	16#00000AD5:
		F_EtherCAT_VendorIDtoString := 'VA Laserautomation GmbH';

	16#00000AD6:
		F_EtherCAT_VendorIDtoString := 'Kleintges Elektrogeratebau GmbH';

	16#00000AD7:
		F_EtherCAT_VendorIDtoString := 'Logosol, Inc.';

	16#00000AD8:
		F_EtherCAT_VendorIDtoString := 'REJ Co., Ltd.';

	16#00000AD9:
		F_EtherCAT_VendorIDtoString := 'TCK Inc.';

	16#00000ADA:
		F_EtherCAT_VendorIDtoString := 'Axetris AG';

	16#00000ADB:
		F_EtherCAT_VendorIDtoString := 'Replicant Automation FZE';

	16#00000ADC:
		F_EtherCAT_VendorIDtoString := 'AIRTEC Pneumatic GmbH';

	16#00000ADD:
		F_EtherCAT_VendorIDtoString := 'Equip-Test Kft.';

	16#00000ADE:
		F_EtherCAT_VendorIDtoString := 'ChromaTan Corporation';

	16#00000ADF:
		F_EtherCAT_VendorIDtoString := 'Ford Motor Company Limited';

	16#00000AE0:
		F_EtherCAT_VendorIDtoString := 'thyssenkrupp Marine Systems GmbH';

	16#00000AE1:
		F_EtherCAT_VendorIDtoString := 'GEFAZ mbH';

	16#00000AE3:
		F_EtherCAT_VendorIDtoString := 'L&T Technology Services Limited';

	16#00000AE5:
		F_EtherCAT_VendorIDtoString := 'The Cyber University of Korea, Department of Mechanical and Control Engineering';

	16#00000AE6:
		F_EtherCAT_VendorIDtoString := 'SCHOBER Elektronik GmbH';

	16#00000AE7:
		F_EtherCAT_VendorIDtoString := 'Simulation and Control Technologies, Inc';

	16#00000AE8:
		F_EtherCAT_VendorIDtoString := 'Guangdong Sumida Automation Co.,Ltd.';

	16#00000AE9:
		F_EtherCAT_VendorIDtoString := 'GEMSS Medical Systems Co.,Ltd.';

	16#00000AEA:
		F_EtherCAT_VendorIDtoString := 'Shanghai Electric Power T&D Group';

	16#00000AEB:
		F_EtherCAT_VendorIDtoString := 'Shandong University, School of Control Science and Engineering';

	16#00000AEC:
		F_EtherCAT_VendorIDtoString := 'Fiessler Elektronik GmbH & Co. KG';

	16#00000AED:
		F_EtherCAT_VendorIDtoString := 'Cencorp Automation Technology Co, Ltd.';

	16#00000AEE:
		F_EtherCAT_VendorIDtoString := 'Venture International Pte Ltd';

	16#00000AEF:
		F_EtherCAT_VendorIDtoString := 'EcoTronic GmbH';

	16#00000AF0:
		F_EtherCAT_VendorIDtoString := 'Shenzhen Donglaier Smart Technology Co., Ltd.';

	16#00000AF1:
		F_EtherCAT_VendorIDtoString := 'Domino UK Limited';

	16#00000AF3:
		F_EtherCAT_VendorIDtoString := 'Elekta Solutions AB';

	16#00000AF4:
		F_EtherCAT_VendorIDtoString := 'Logic Fruit Technologies Pvt. Ltd.';

	16#00000AF5:
		F_EtherCAT_VendorIDtoString := 'ecocoach AG';

	16#00000AF6:
		F_EtherCAT_VendorIDtoString := 'SIOS Metechnik GmbH';

	16#00000AF7:
		F_EtherCAT_VendorIDtoString := 'Jabil Circuit Magyarorszag Kft.';

	16#00000AF8:
		F_EtherCAT_VendorIDtoString := 'seven dreamers laundroid, inc.';

	16#00000AF9:
		F_EtherCAT_VendorIDtoString := 'VR Group, a.s.';

	16#00000AFA:
		F_EtherCAT_VendorIDtoString := 'Afag Automation AG';

	16#00000AFB:
		F_EtherCAT_VendorIDtoString := 'Miyagi Nikon Precision Co., Ltd.';

	16#00000AFC:
		F_EtherCAT_VendorIDtoString := 'AutomationWare S.r.l.';

	16#00000AFD:
		F_EtherCAT_VendorIDtoString := 'Isar Aerospace Technologies GmbH';

	16#00000AFE:
		F_EtherCAT_VendorIDtoString := 'GTSystem GmbH';

	16#00000AFF:
		F_EtherCAT_VendorIDtoString := 'Technische Universitat Munchen, Department of Physics';

	16#00000B00:
		F_EtherCAT_VendorIDtoString := 'S+S Regeltechnik GmbH';

	16#00000B01:
		F_EtherCAT_VendorIDtoString := 'Osaka University, Graduate School of Engineering Science';

	16#00000B02:
		F_EtherCAT_VendorIDtoString := 'Vogtlin Instruments GmbH';

	16#00000B03:
		F_EtherCAT_VendorIDtoString := 'TOHAN DENSHI KIKI CO.,LTD.';

	16#00000B04:
		F_EtherCAT_VendorIDtoString := 'Shinwa Industries, Inc.';

	16#00000B05:
		F_EtherCAT_VendorIDtoString := 'Suzhou Linkhou Robot Co.,Ltd';

	16#00000B06:
		F_EtherCAT_VendorIDtoString := 'DMC, Inc.';

	16#00000B07:
		F_EtherCAT_VendorIDtoString := 'Nippon Pulse Motor Co., Ltd.';

	16#00000B08:
		F_EtherCAT_VendorIDtoString := 'LANG GmbH & Co. KG';

	16#00000B09:
		F_EtherCAT_VendorIDtoString := 'STICHT Technologie GmbH';

	16#00000B0A:
		F_EtherCAT_VendorIDtoString := 'HIMS Co., Ltd.';

	16#00000B0B:
		F_EtherCAT_VendorIDtoString := 'WITRON Logistik + Informatik GmbH';

	16#00000B0C:
		F_EtherCAT_VendorIDtoString := 'Vistec Electron Beam GmbH';

	16#00000B0D:
		F_EtherCAT_VendorIDtoString := 'General Atomics';

	16#00000B0E:
		F_EtherCAT_VendorIDtoString := 'Teubner Industrie-Elektronik GmbH';

	16#00000B0F:
		F_EtherCAT_VendorIDtoString := 'DEWETRON GmbH';

	16#00000B10:
		F_EtherCAT_VendorIDtoString := 'Philip Morris Products SA';

	16#00000B11:
		F_EtherCAT_VendorIDtoString := 'Nihon Protech Software Co., Ltd.';

	16#00000B13:
		F_EtherCAT_VendorIDtoString := 'Industrial Indexing Systems, Inc.';

	16#00000B14:
		F_EtherCAT_VendorIDtoString := 'AKIM METAL Sanayi Ve Ticaret Anonim Sirketi';

	16#00000B15:
		F_EtherCAT_VendorIDtoString := 'MEODAT Messtechnik, Ortung und Datenverarbeitung GmbH';

	16#00000B17:
		F_EtherCAT_VendorIDtoString := 'Goyo Electronics Co.,Ltd.';

	16#00000B18:
		F_EtherCAT_VendorIDtoString := 'Shanghai Golytec Automation Co., Ltd.';

	16#00000B19:
		F_EtherCAT_VendorIDtoString := 'Redcur GmbH';

	16#00000B1A:
		F_EtherCAT_VendorIDtoString := 'Room3327, Inc.';

	16#00000B1C:
		F_EtherCAT_VendorIDtoString := 'Love Electronics Ltd';

	16#00000B1D:
		F_EtherCAT_VendorIDtoString := 'Fontys University of Applied Sciences, School of Information & Communication Technology';

	16#00000B1E:
		F_EtherCAT_VendorIDtoString := 'Hocoma AG';

	16#00000B1F:
		F_EtherCAT_VendorIDtoString := 'Sensor Instruments Entwicklungs- und Vertriebs-GmbH';

	16#00000B20:
		F_EtherCAT_VendorIDtoString := 'Reboocon Bionics B.V.';

	16#00000B21:
		F_EtherCAT_VendorIDtoString := 'Evident Canada Inc.';

	16#00000B22:
		F_EtherCAT_VendorIDtoString := 'Photon Control Inc.';

	16#00000B23:
		F_EtherCAT_VendorIDtoString := 'NK Labs, LLC';

	16#00000B24:
		F_EtherCAT_VendorIDtoString := 'Excelpoint Systems (India) Pvt Ltd';

	16#00000B25:
		F_EtherCAT_VendorIDtoString := '"Gheorghe Asachi" Technical University of Iasi, Faculty of Automatic Control and Computer Engineering';

	16#00000B26:
		F_EtherCAT_VendorIDtoString := 'Manroland Sheetfed GmbH';

	16#00000B27:
		F_EtherCAT_VendorIDtoString := 'OPTEX FA CO., LTD.';

	16#00000B28:
		F_EtherCAT_VendorIDtoString := 'SMAC Corporation';

	16#00000B2A:
		F_EtherCAT_VendorIDtoString := 'SAITEL S.r.l.';

	16#00000B2B:
		F_EtherCAT_VendorIDtoString := 'Hebi Haichang Special Equipment Co.,Ltd.';

	16#00000B2C:
		F_EtherCAT_VendorIDtoString := 'Salunda Ltd';

	16#00000B2D:
		F_EtherCAT_VendorIDtoString := 'Higerman CNC Technology (SZ) Limited';

	16#00000B2E:
		F_EtherCAT_VendorIDtoString := 'IPG Laser GmbH & Co. KG';

	16#00000B2F:
		F_EtherCAT_VendorIDtoString := 'RTSoft, AO';

	16#00000B30:
		F_EtherCAT_VendorIDtoString := 'Dalian Hi-Sensor Technology Co., Ltd.';

	16#00000B31:
		F_EtherCAT_VendorIDtoString := 'alpiscan srls';

	16#00000B32:
		F_EtherCAT_VendorIDtoString := 'DYNAMIC OPTICS s.r.l.';

	16#00000B33:
		F_EtherCAT_VendorIDtoString := 'OOO “ITS-Sibir”';

	16#00000B34:
		F_EtherCAT_VendorIDtoString := 'SUMITOMO RIKO Company Limited';

	16#00000B35:
		F_EtherCAT_VendorIDtoString := 'Tianjin Automa Technology Co. Ltd.';

	16#00000B37:
		F_EtherCAT_VendorIDtoString := 'Human Automation Co., Ltd.';

	16#00000B38:
		F_EtherCAT_VendorIDtoString := 'Aplex Technology Inc.';

	16#00000B39:
		F_EtherCAT_VendorIDtoString := 'Shanghai Jesee Auto System Co., Ltd';

	16#00000B3A:
		F_EtherCAT_VendorIDtoString := 'Kunming Unionscience Technology Co.,Ltd';

	16#00000B3B:
		F_EtherCAT_VendorIDtoString := 'Fitz-Thors Engineering, Inc.';

	16#00000B3C:
		F_EtherCAT_VendorIDtoString := 'ACTIA Automotive SA';

	16#00000B3D:
		F_EtherCAT_VendorIDtoString := 'Kunshan SVL Electric Co.,Ltd';

	16#00000B3E:
		F_EtherCAT_VendorIDtoString := 'SilCore Technology';

	16#00000B3F:
		F_EtherCAT_VendorIDtoString := 'SHENZHEN QITAI TECHNOLOGY CO.LTD';

	16#00000B40:
		F_EtherCAT_VendorIDtoString := 'A. Sturzenegger Elektronik GmbH';

	16#00000B41:
		F_EtherCAT_VendorIDtoString := 'ZEUS CO., LTD.';

	16#00000B42:
		F_EtherCAT_VendorIDtoString := 'BETAMONT s.r.o.';

	16#00000B43:
		F_EtherCAT_VendorIDtoString := 'Strategy Automation S.r.l.';

	16#00000B44:
		F_EtherCAT_VendorIDtoString := 'Fachhochschule Nordwestschweiz, Hochschule fur Technik, Institut fur Automation';

	16#00000B45:
		F_EtherCAT_VendorIDtoString := 'SMS group GmbH';

	16#00000B46:
		F_EtherCAT_VendorIDtoString := 'TRUMPF Schweiz AG';

	16#00000B47:
		F_EtherCAT_VendorIDtoString := 'Fraunhofer-Institut fur Silicatforschung ISC';

	16#00000B48:
		F_EtherCAT_VendorIDtoString := 'The University of Tokyo, Graduate School of Information Science and Technology';

	16#00000B49:
		F_EtherCAT_VendorIDtoString := 'Indian Institute of Science, Interdisciplinary Centre for Energy Research';

	16#00000B4A:
		F_EtherCAT_VendorIDtoString := 'Overlay Technology OU';

	16#00000B4B:
		F_EtherCAT_VendorIDtoString := 'CK Automation, LLC';

	16#00000B4D:
		F_EtherCAT_VendorIDtoString := 'OOO "Kompex-T"';

	16#00000B4E:
		F_EtherCAT_VendorIDtoString := 'Ostbayerische Technische Hochschule Regensburg, Fakultat Maschinenbau';

	16#00000B4F:
		F_EtherCAT_VendorIDtoString := 'Hefei Eagle Automation Engineering Technology Co., Ltd.';

	16#00000B50:
		F_EtherCAT_VendorIDtoString := 'Vertiv Tech Co., Ltd';

	16#00000B51:
		F_EtherCAT_VendorIDtoString := 'Sanying MotionControl Instruments Ltd.';

	16#00000B52:
		F_EtherCAT_VendorIDtoString := 'Jiangsu Saiyang Mechanical & Electrical Technology Co., Ltd.';

	16#00000B53:
		F_EtherCAT_VendorIDtoString := 'Robosoft NV';

	16#00000B54:
		F_EtherCAT_VendorIDtoString := 'MotionBank';

	16#00000B55:
		F_EtherCAT_VendorIDtoString := 'South China University of Technology, School of Automation Science & Engineering';

	16#00000B56:
		F_EtherCAT_VendorIDtoString := 'Oetiker Schweiz AG';

	16#00000B57:
		F_EtherCAT_VendorIDtoString := 'Chiang Mai University, Faculty of Engineering';

	16#00000B58:
		F_EtherCAT_VendorIDtoString := 'Shenzhen FOXON Automation Technology Co., Ltd.';

	16#00000B59:
		F_EtherCAT_VendorIDtoString := 'Heinmade BV';

	16#00000B5A:
		F_EtherCAT_VendorIDtoString := 'ING-AUTOMATION';

	16#00000B5B:
		F_EtherCAT_VendorIDtoString := 'Vanteon Corporation';

	16#00000B5C:
		F_EtherCAT_VendorIDtoString := 'Solvine, Inc.';

	16#00000B5D:
		F_EtherCAT_VendorIDtoString := 'SHINWA Controls Co., Ltd.';

	16#00000B5E:
		F_EtherCAT_VendorIDtoString := 'Sierra CP Engineering Ltd.';

	16#00000B5F:
		F_EtherCAT_VendorIDtoString := 'Rope Robotics ApS';

	16#00000B60:
		F_EtherCAT_VendorIDtoString := 'Hefei Sineva Intelligent Machine Co.,Ltd';

	16#00000B61:
		F_EtherCAT_VendorIDtoString := 'Shenzhen Porcheson Technology Co., Ltd';

	16#00000B62:
		F_EtherCAT_VendorIDtoString := 'Greenlight Innovation Inc.';

	16#00000B63:
		F_EtherCAT_VendorIDtoString := 'PCB Piezotronics, Inc.';

	16#00000B64:
		F_EtherCAT_VendorIDtoString := 'microGauge AG';

	16#00000B65:
		F_EtherCAT_VendorIDtoString := 'EL Klaszter Iroda Kft.';

	16#00000B66:
		F_EtherCAT_VendorIDtoString := 'A.B.Esse Spa';

	16#00000B67:
		F_EtherCAT_VendorIDtoString := 'Corindus, Inc.';

	16#00000B68:
		F_EtherCAT_VendorIDtoString := 'Celeroton AG';

	16#00000B69:
		F_EtherCAT_VendorIDtoString := 'SAMHYUN Co. Ltd.';

	16#00000B6A:
		F_EtherCAT_VendorIDtoString := 'Ecole Polytechnique Federale de Lausanne, School of Basic Sciences';

	16#00000B6B:
		F_EtherCAT_VendorIDtoString := 'AVIC-XINHANG YUBEI STEERING SYSTEM (XINXIANG) CO.,LTD';

	16#00000B6C:
		F_EtherCAT_VendorIDtoString := 'Creative Conners, Inc.';

	16#00000B6D:
		F_EtherCAT_VendorIDtoString := 'Mamezou Co.,Ltd.';

	16#00000B6E:
		F_EtherCAT_VendorIDtoString := 'Raith B.V.';

	16#00000B6F:
		F_EtherCAT_VendorIDtoString := 'Soft Harmony';

	16#00000B70:
		F_EtherCAT_VendorIDtoString := 'Elektrik Uretim A.S.';

	16#00000B71:
		F_EtherCAT_VendorIDtoString := 'Delft University of Technology, Electronic and Mechanical Support Division (DEMO)';

	16#00000B72:
		F_EtherCAT_VendorIDtoString := 'machineering GmbH & Co. KG';

	16#00000B73:
		F_EtherCAT_VendorIDtoString := 'GRAPHIMECC S.r.l.';

	16#00000B74:
		F_EtherCAT_VendorIDtoString := 'TOPTICA Projects GmbH';

	16#00000B75:
		F_EtherCAT_VendorIDtoString := 'Enlaica Co., Ltd.';

	16#00000B76:
		F_EtherCAT_VendorIDtoString := 'SYSTEC Corporation';

	16#00000B77:
		F_EtherCAT_VendorIDtoString := 'Sherpa Inc.';

	16#00000B78:
		F_EtherCAT_VendorIDtoString := 'Sioux Embedded Systems B.V.';

	16#00000B79:
		F_EtherCAT_VendorIDtoString := 'UNISEM Co., Ltd.';

	16#00000B7A:
		F_EtherCAT_VendorIDtoString := 'William Petersen Elektronik A/S';

	16#00000B7B:
		F_EtherCAT_VendorIDtoString := 'Shanghai Velle Automobile Air Conditioner Co., Ltd.';

	16#00000B7C:
		F_EtherCAT_VendorIDtoString := 'Vision Tech Co.';

	16#00000B7D:
		F_EtherCAT_VendorIDtoString := 'Technische Universitat Wien, Fakultat fur Elektrotechnik und Informationstechnik';

	16#00000B7E:
		F_EtherCAT_VendorIDtoString := 'Universitat Augsburg, Fakultat fur Angewandte Informatik';

	16#00000B7F:
		F_EtherCAT_VendorIDtoString := 'Tecnomotion Srl';

	16#00000B80:
		F_EtherCAT_VendorIDtoString := 'Microservo Co., Ltd.';

	16#00000B81:
		F_EtherCAT_VendorIDtoString := 'Micro CleanRoom Technology GmbH';

	16#00000B82:
		F_EtherCAT_VendorIDtoString := 'Global Motion & Systems Inc.';

	16#00000B83:
		F_EtherCAT_VendorIDtoString := 'L3 Technologies, Datron Advanced Technologies';

	16#00000B84:
		F_EtherCAT_VendorIDtoString := 'NTN Technical Service Corporation';

	16#00000B85:
		F_EtherCAT_VendorIDtoString := 'Chugoku Electric Manufacturing Co.,Inc.';

	16#00000B86:
		F_EtherCAT_VendorIDtoString := 'European Spallation Source ERIC, Integrated Control System Division';

	16#00000B87:
		F_EtherCAT_VendorIDtoString := 'MARS CO., LTD.';

	16#00000B88:
		F_EtherCAT_VendorIDtoString := 'SCOPX LABS';

	16#00000B89:
		F_EtherCAT_VendorIDtoString := 'Laser Mechanisms, Inc.';

	16#00000B8A:
		F_EtherCAT_VendorIDtoString := 'TechnoPro, Inc.';

	16#00000B8B:
		F_EtherCAT_VendorIDtoString := 'Advanced Micro Controls, Inc.';

	16#00000B8C:
		F_EtherCAT_VendorIDtoString := 'Intelligence Technology of CEC Co., Ltd';

	16#00000B8D:
		F_EtherCAT_VendorIDtoString := 'Applied Dynamics International, Inc.';

	16#00000B8E:
		F_EtherCAT_VendorIDtoString := 'Conch Electronic Co.,Ltd.';

	16#00000B8F:
		F_EtherCAT_VendorIDtoString := 'Shenzhen Lisan M&E Co., Ltd.';

	16#00000B90:
		F_EtherCAT_VendorIDtoString := 'FOXIDE LLC';

	16#00000B91:
		F_EtherCAT_VendorIDtoString := 'C2P Inc.';

	16#00000B92:
		F_EtherCAT_VendorIDtoString := 'SonMicroSystem Co.';

	16#00000B94:
		F_EtherCAT_VendorIDtoString := 'HUST Automation System Co., Ltd.';

	16#00000B95:
		F_EtherCAT_VendorIDtoString := 'ASIX Electronics Corporation';

	16#00000B97:
		F_EtherCAT_VendorIDtoString := 'Laboratoire dAnalyse et dArchitecture des Systemes (LAAS-CNRS)';

	16#00000B98:
		F_EtherCAT_VendorIDtoString := 'KM DIGITECH CO., LTD.';

	16#00000B99:
		F_EtherCAT_VendorIDtoString := 'Sens4 A/S';

	16#00000B9A:
		F_EtherCAT_VendorIDtoString := 'Nidec Research and Development Center, Taiwan';

	16#00000B9D:
		F_EtherCAT_VendorIDtoString := 'Cajo Technologies Oy';

	16#00000B9E:
		F_EtherCAT_VendorIDtoString := 'VAS HIGH TECHNOLOGY SOLUTION CORPORATION';

	16#00000B9F:
		F_EtherCAT_VendorIDtoString := 'Beijing Chymotion Control Technology Co. Ltd';

	16#00000BA0:
		F_EtherCAT_VendorIDtoString := 'MarquipWardUnited';

	16#00000BA1:
		F_EtherCAT_VendorIDtoString := 'Komax Singapore Pte Ltd';

	16#00000BA2:
		F_EtherCAT_VendorIDtoString := 'Persimmon Technologies Corporation';

	16#00000BA3:
		F_EtherCAT_VendorIDtoString := 'Tohoku University, New Industry Creation Hatchery Center (NICHe), Fluctuation Free Facility (FFF)';

	16#00000BA4:
		F_EtherCAT_VendorIDtoString := 'Rheinische Fachhochschule Koln gGmbH, Ingenieurwesen';

	16#00000BA5:
		F_EtherCAT_VendorIDtoString := 'Luminize';

	16#00000BA6:
		F_EtherCAT_VendorIDtoString := 'v6e Limited';

	16#00000BA7:
		F_EtherCAT_VendorIDtoString := 'ECA ROBOTICS SASU';

	16#00000BA8:
		F_EtherCAT_VendorIDtoString := 'Sphere Fluidics Limited';

	16#00000BA9:
		F_EtherCAT_VendorIDtoString := 'WELCON Systems Inc.';

	16#00000BAA:
		F_EtherCAT_VendorIDtoString := 'Exor International S.p.A';

	16#00000BAB:
		F_EtherCAT_VendorIDtoString := 'Dekimo Turnhout';

	16#00000BAC:
		F_EtherCAT_VendorIDtoString := 'Lavender CE Pty Ltd';

	16#00000BAD:
		F_EtherCAT_VendorIDtoString := 'Science in Motion Technology Corporation, Ltd.';

	16#00000BAE:
		F_EtherCAT_VendorIDtoString := 'IST Ingenieurburo fur Sensortechnik GmbH';

	16#00000BAF:
		F_EtherCAT_VendorIDtoString := 'maku engineering GmbH';

	16#00000BB0:
		F_EtherCAT_VendorIDtoString := 'Geoservices Equipements SAS';

	16#00000BB1:
		F_EtherCAT_VendorIDtoString := 'NEST Electronics GmbH';

	16#00000BB2:
		F_EtherCAT_VendorIDtoString := 'MR Shim GmbH';

	16#00000BB4:
		F_EtherCAT_VendorIDtoString := 'Zettaone Technologies India Pvt Ltd';

	16#00000BB6:
		F_EtherCAT_VendorIDtoString := 'Universitat Augsburg, Fakultat fur angewandte Informatik, Institut fur Informatik';

	16#00000BB7:
		F_EtherCAT_VendorIDtoString := 'SCHUNK Electronic Solutions GmbH';

	16#00000BB8:
		F_EtherCAT_VendorIDtoString := 'KOORD Sarl';

	16#00000BB9:
		F_EtherCAT_VendorIDtoString := 'regenHU Ltd.';

	16#00000BBA:
		F_EtherCAT_VendorIDtoString := 'VONSCH spol. s r.o.';

	16#00000BBC:
		F_EtherCAT_VendorIDtoString := 'Bore Automation Tech. Co., Ltd.';

	16#00000BBD:
		F_EtherCAT_VendorIDtoString := 'Board Planning Co., Ltd.';

	16#00000BBE:
		F_EtherCAT_VendorIDtoString := 'Kamp & Kotter GmbH';

	16#00000BBF:
		F_EtherCAT_VendorIDtoString := 'IOTech Systems Limited';

	16#00000BC0:
		F_EtherCAT_VendorIDtoString := 'Altinay Robot Technologies Inc.';

	16#00000BC1:
		F_EtherCAT_VendorIDtoString := 'Lorenz Messtechnik GmbH';

	16#00000BC2:
		F_EtherCAT_VendorIDtoString := 'LJ Welding Automation';

	16#00000BC3:
		F_EtherCAT_VendorIDtoString := 'DMP Electronics Inc.';

	16#00000BC4:
		F_EtherCAT_VendorIDtoString := 'Dima Motor Tec. Co., Ltd.';

	16#00000BC5:
		F_EtherCAT_VendorIDtoString := 'Fraunhofer-Institut fur Produktionstechnik und Automatisierung';

	16#00000BC6:
		F_EtherCAT_VendorIDtoString := 'Schneider Electric (China) Co., Ltd.';

	16#00000BC7:
		F_EtherCAT_VendorIDtoString := 'Suzhou DaFang Special Vehicle Co., Ltd';

	16#00000BC8:
		F_EtherCAT_VendorIDtoString := 'Shenzhen OUYE Intelligent Technology Co., Ltd';

	16#00000BC9:
		F_EtherCAT_VendorIDtoString := 'HBH Microwave GmbH';

	16#00000BCA:
		F_EtherCAT_VendorIDtoString := 'MTA B.V.';

	16#00000BCB:
		F_EtherCAT_VendorIDtoString := 'SYSTEM ARTWARE, Inc.';

	16#00000BCC:
		F_EtherCAT_VendorIDtoString := 'ProDSP Technologies Zrt.';

	16#00000BCD:
		F_EtherCAT_VendorIDtoString := 'Hypersen Technologies Co., Ltd';

	16#00000BCE:
		F_EtherCAT_VendorIDtoString := 'Pyramid Vacuum LLC';

	16#00000BCF:
		F_EtherCAT_VendorIDtoString := 'Hanbaek Tech Co., Ltd.';

	16#00000BD0:
		F_EtherCAT_VendorIDtoString := 'SC3 Automation Inc.';

	16#00000BD1:
		F_EtherCAT_VendorIDtoString := 'Fachhochschule Nordwestschweiz, Hochschule fur Technik, Institut fur Sensorik und Elektronik';

	16#00000BD2:
		F_EtherCAT_VendorIDtoString := 'innofas GmbH';

	16#00000BD3:
		F_EtherCAT_VendorIDtoString := 'Orbray Co., Ltd.';

	16#00000BD4:
		F_EtherCAT_VendorIDtoString := 'YUNNAN KSEC INTELLIGENT EQUIPMENT CO.,LTD.';

	16#00000BD6:
		F_EtherCAT_VendorIDtoString := 'Industrial Solutions Zuid-Oost B.V. (Actemium Electronics)';

	16#00000BD7:
		F_EtherCAT_VendorIDtoString := 'BETONMAC S.A.';

	16#00000BD8:
		F_EtherCAT_VendorIDtoString := 'Manufacturing Objects';

	16#00000BD9:
		F_EtherCAT_VendorIDtoString := 'Chen Yuan International Co., Ltd.';

	16#00000BDB:
		F_EtherCAT_VendorIDtoString := 'Griffin Technology Co., Ltd.';

	16#00000BDC:
		F_EtherCAT_VendorIDtoString := 'RORZE CORPORATION';

	16#00000BDD:
		F_EtherCAT_VendorIDtoString := 'Bruker Daltonik GmbH';

	16#00000BDE:
		F_EtherCAT_VendorIDtoString := 'Logos01 Srl';

	16#00000BDF:
		F_EtherCAT_VendorIDtoString := 'Coaters Paradise GmbH';

	16#00000BE0:
		F_EtherCAT_VendorIDtoString := 'Hahn-Schickard-Gesellschaft fur angewandte Forschung e.V.';

	16#00000BE2:
		F_EtherCAT_VendorIDtoString := 'R&D Company "Vector" LLC';

	16#00000BE3:
		F_EtherCAT_VendorIDtoString := 'ReeR SpA';

	16#00000BE4:
		F_EtherCAT_VendorIDtoString := 'HP Scitex Ltd.';

	16#00000BE5:
		F_EtherCAT_VendorIDtoString := 'Hitachi Automotive Systems Americas, Inc.';

	16#00000BE6:
		F_EtherCAT_VendorIDtoString := 'Zhejiang Eternal Automation Sci-Tec Co.,Ltd';

	16#00000BE7:
		F_EtherCAT_VendorIDtoString := 'Shenzhen Siron Electrical Co.,Ltd.';

	16#00000BE8:
		F_EtherCAT_VendorIDtoString := 'ARUP Laboratories';

	16#00000BE9:
		F_EtherCAT_VendorIDtoString := 'LETech Co.,Ltd.';

	16#00000BEA:
		F_EtherCAT_VendorIDtoString := 'Bangkok University, School of Engineering, Robotics Laboratory';

	16#00000BEB:
		F_EtherCAT_VendorIDtoString := 'Kontron Electronics GmbH';

	16#00000BEC:
		F_EtherCAT_VendorIDtoString := 'Shanghai Junqian Sensing Technology Co., Ltd.';

	16#00000BEE:
		F_EtherCAT_VendorIDtoString := 'VI.BE.MAC s.p.a.';

	16#00000BEF:
		F_EtherCAT_VendorIDtoString := 'EMG Automation GmbH';

	16#00000BF0:
		F_EtherCAT_VendorIDtoString := 'American Controls & Automation, Inc.';

	16#00000BF1:
		F_EtherCAT_VendorIDtoString := 'Ascale Enterprise Co., Ltd.';

	16#00000BF2:
		F_EtherCAT_VendorIDtoString := 'University of Applied Sciences and Arts Western Switzerland (HES-SO Fribourg)';

	16#00000BF3:
		F_EtherCAT_VendorIDtoString := 'Lantronix, Inc.';

	16#00000BF4:
		F_EtherCAT_VendorIDtoString := 'Technische Hochschule Rosenheim';

	16#00000BF5:
		F_EtherCAT_VendorIDtoString := 'LEIFERT INDUCTION GmbH';

	16#00000BF6:
		F_EtherCAT_VendorIDtoString := 'Automation of Things Europe GmbH';

	16#00000BF7:
		F_EtherCAT_VendorIDtoString := 'SAMWON ACT Co.,Ltd';

	16#00000BF8:
		F_EtherCAT_VendorIDtoString := 'Wenling Yuhai Electromechanical CO.,LTD';

	16#00000BF9:
		F_EtherCAT_VendorIDtoString := 'Faraday Motion Controls Ltd.';

	16#00000BFA:
		F_EtherCAT_VendorIDtoString := 'Nikon Systems Inc.';

	16#00000BFB:
		F_EtherCAT_VendorIDtoString := 'Sanitas EG S.r.l.';

	16#00000BFC:
		F_EtherCAT_VendorIDtoString := 'Videojet Technologies Inc.';

	16#00000BFD:
		F_EtherCAT_VendorIDtoString := 'ABB AG';

	16#00000BFE:
		F_EtherCAT_VendorIDtoString := 'WARDJet LLC';

	16#00000BFF:
		F_EtherCAT_VendorIDtoString := 'Ichor Systems, Inc.';

	16#00000C00:
		F_EtherCAT_VendorIDtoString := 'UTAREX Co., Ltd.';

	16#00000C01:
		F_EtherCAT_VendorIDtoString := 'GAON SOLUTION Ltd.';

	16#00000C02:
		F_EtherCAT_VendorIDtoString := 'Highlight Tech Corp.';

	16#00000C03:
		F_EtherCAT_VendorIDtoString := 'PO OWEN LLC';

	16#00000C04:
		F_EtherCAT_VendorIDtoString := 'RFPT Co., Ltd.';

	16#00000C05:
		F_EtherCAT_VendorIDtoString := 'Roboteq, Inc.';

	16#00000C06:
		F_EtherCAT_VendorIDtoString := 'Norgren Manufacturing Co., Ltd.';

	16#00000C07:
		F_EtherCAT_VendorIDtoString := 'FarmWise Labs, Inc.';

	16#00000C08:
		F_EtherCAT_VendorIDtoString := 'AŽD Praha s.r.o.';

	16#00000C0A:
		F_EtherCAT_VendorIDtoString := 'Can Man AG';

	16#00000C0B:
		F_EtherCAT_VendorIDtoString := 'Plustherm Point AG';

	16#00000C0C:
		F_EtherCAT_VendorIDtoString := 'MinebeaMitsumi Inc.';

	16#00000C0D:
		F_EtherCAT_VendorIDtoString := 'System Level Solutions (India) Pvt. Ltd.';

	16#00000C0E:
		F_EtherCAT_VendorIDtoString := 'EverMAX s.r.o.';

	16#00000C0F:
		F_EtherCAT_VendorIDtoString := 'Maruyama Manufacturing Corporation (DBA Maruyama Chillers Corporation)';

	16#00000C10:
		F_EtherCAT_VendorIDtoString := 'Han’s Assembly and Testing Technology (Singapore) Pte. Ltd.';

	16#00000C11:
		F_EtherCAT_VendorIDtoString := 'Cordova Industrial Integradores S.A. de C.V.';

	16#00000C12:
		F_EtherCAT_VendorIDtoString := 'NAMOO Co., Ltd.';

	16#00000C13:
		F_EtherCAT_VendorIDtoString := 'Blu Technology di Ing Carlo Mauri';

	16#00000C14:
		F_EtherCAT_VendorIDtoString := 'isel Germany AG';

	16#00000C15:
		F_EtherCAT_VendorIDtoString := 'UNITEK Industrie Elektronik GmbH';

	16#00000C16:
		F_EtherCAT_VendorIDtoString := 'Tohan-Engineering Corporation';

	16#00000C17:
		F_EtherCAT_VendorIDtoString := 'Machine Prognostics AS';

	16#00000C18:
		F_EtherCAT_VendorIDtoString := 'Avestron Inc.';

	16#00000C19:
		F_EtherCAT_VendorIDtoString := 'AP Systems Co., Ltd.';

	16#00000C1A:
		F_EtherCAT_VendorIDtoString := 'TIAN JIN SUNKE DIGITAL CONTROL TECHNOLOGY CO.,LTD';

	16#00000C1B:
		F_EtherCAT_VendorIDtoString := 'Robotech Co., Ltd.';

	16#00000C1C:
		F_EtherCAT_VendorIDtoString := 'AccuteX Technologies Co., Ltd.';

	16#00000C1D:
		F_EtherCAT_VendorIDtoString := 'Coherent Mainz (DILAS Diodenlaser GmbH)';

	16#00000C1E:
		F_EtherCAT_VendorIDtoString := 'Daxta Equipamentos Eletronicos Industria e Comercio Ltda';

	16#00000C20:
		F_EtherCAT_VendorIDtoString := 'ADG Automatisierung Dresden GmbH';

	16#00000C21:
		F_EtherCAT_VendorIDtoString := 'WHITEvoid GmbH';

	16#00000C22:
		F_EtherCAT_VendorIDtoString := 'BAS BV';

	16#00000C23:
		F_EtherCAT_VendorIDtoString := 'RS Elektroniksysteme GmbH';

	16#00000C25:
		F_EtherCAT_VendorIDtoString := 'HORIBA FuelCon GmbH';

	16#00000C26:
		F_EtherCAT_VendorIDtoString := 'miCos Iberia S.L.';

	16#00000C27:
		F_EtherCAT_VendorIDtoString := 'Slovak Academy of Sciences, Institute of Electrical Engineering';

	16#00000C28:
		F_EtherCAT_VendorIDtoString := 'Roketsan A.S.';

	16#00000C29:
		F_EtherCAT_VendorIDtoString := 'Bescom Global Co., Ltd.';

	16#00000C2A:
		F_EtherCAT_VendorIDtoString := 'Magnet-Schultz GmbH & Co. KG';

	16#00000C2B:
		F_EtherCAT_VendorIDtoString := 'NEWSUBSTANCE Limited';

	16#00000C2C:
		F_EtherCAT_VendorIDtoString := 'JingQi (Tianjin) Technology Co., Ltd.';

	16#00000C2D:
		F_EtherCAT_VendorIDtoString := 'TSK Prufsysteme GmbH';

	16#00000C2E:
		F_EtherCAT_VendorIDtoString := 'Airity Technologies, Inc.';

	16#00000C2F:
		F_EtherCAT_VendorIDtoString := 'EEP Elektro Elektronik Pranjic GmbH';

	16#00000C30:
		F_EtherCAT_VendorIDtoString := 'MovekoTech Oy';

	16#00000C31:
		F_EtherCAT_VendorIDtoString := 'Federal State Institution "Scientific Research Institute for System Analysis of the Russian Academy of Sciences"';

	16#00000C32:
		F_EtherCAT_VendorIDtoString := 'Nearfield Instruments B.V.';

	16#00000C33:
		F_EtherCAT_VendorIDtoString := 'TUBITAK BILGEM, National Research Institute of Electronics and Cryptology (UEKAE)';

	16#00000C34:
		F_EtherCAT_VendorIDtoString := 'Siemens Energy Global GmbH & Co. KG';

	16#00000C35:
		F_EtherCAT_VendorIDtoString := 'progress Maschinen & Automation AG';

	16#00000C36:
		F_EtherCAT_VendorIDtoString := 'Heliotis AG';

	16#00000C37:
		F_EtherCAT_VendorIDtoString := 'Strong Plus Technology GmbH';

	16#00000C38:
		F_EtherCAT_VendorIDtoString := 'LS Energy Solutions LLC';

	16#00000C39:
		F_EtherCAT_VendorIDtoString := 'Yaskawa Controls Co., Ltd.';

	16#00000C3A:
		F_EtherCAT_VendorIDtoString := 'NOVUSS-Automation GmbH';

	16#00000C3C:
		F_EtherCAT_VendorIDtoString := 'Sanwa Engineering Corp.';

	16#00000C3D:
		F_EtherCAT_VendorIDtoString := 'WIBOND Informationssysteme GmbH';

	16#00000C3E:
		F_EtherCAT_VendorIDtoString := 'MSP, a division of TSI Inc.';

	16#00000C3F:
		F_EtherCAT_VendorIDtoString := 'Wuxi Xinchang Electronic Technology Co., Ltd.';

	16#00000C40:
		F_EtherCAT_VendorIDtoString := 'NDK Semiconductor Co., Ltd.';

	16#00000C41:
		F_EtherCAT_VendorIDtoString := 'MS Ultraschall Technologie GmbH';

	16#00000C42:
		F_EtherCAT_VendorIDtoString := 'Korea University of Technology and Education (KOREATECH)';

	16#00000C43:
		F_EtherCAT_VendorIDtoString := 'Accelerated Software Engineering Ltd.';

	16#00000C44:
		F_EtherCAT_VendorIDtoString := 'Shenzhen Instar Electromechanical Technology Development Co., Ltd.';

	16#00000C45:
		F_EtherCAT_VendorIDtoString := 'Redler Technologies Ltd.';

	16#00000C46:
		F_EtherCAT_VendorIDtoString := 'NPOOO "Sital"';

	16#00000C47:
		F_EtherCAT_VendorIDtoString := 'Eaton Corporation';

	16#00000C48:
		F_EtherCAT_VendorIDtoString := 'Techservo (Shenzhen) Co., Ltd.';

	16#00000C49:
		F_EtherCAT_VendorIDtoString := 'Fabmatics GmbH';

	16#00000C4A:
		F_EtherCAT_VendorIDtoString := 'Sasaki Sekkei Co., Ltd.';

	16#00000C4B:
		F_EtherCAT_VendorIDtoString := 'Lohnert Elektronik GmbH';

	16#00000C4C:
		F_EtherCAT_VendorIDtoString := 'Vendee Concept SA';

	16#00000C4D:
		F_EtherCAT_VendorIDtoString := 'Nobleo Technology Holding BV';

	16#00000C4E:
		F_EtherCAT_VendorIDtoString := 'ECI Technology, Inc.';

	16#00000C4F:
		F_EtherCAT_VendorIDtoString := 'Linus G Productions GmbH';

	16#00000C50:
		F_EtherCAT_VendorIDtoString := 'PCB Elektronik San. Ve Tic. Ltd. Sti.';

	16#00000C51:
		F_EtherCAT_VendorIDtoString := 'Omron Scientific Technologies, Inc.';

	16#00000C52:
		F_EtherCAT_VendorIDtoString := 'Engineered Arts Limited';

	16#00000C53:
		F_EtherCAT_VendorIDtoString := 'NASA Jet Propulsion Laboratory';

	16#00000C54:
		F_EtherCAT_VendorIDtoString := 'Accelovant Technologies Corporation';

	16#00000C55:
		F_EtherCAT_VendorIDtoString := 'Hirata Corporation';

	16#00000C56:
		F_EtherCAT_VendorIDtoString := 'Fujian Nebula Electronics Co.,Ltd.';

	16#00000C57:
		F_EtherCAT_VendorIDtoString := 'Test Research, Inc.';

	16#00000C58:
		F_EtherCAT_VendorIDtoString := 'CYSCO Co., Ltd.';

	16#00000C59:
		F_EtherCAT_VendorIDtoString := 'Esko-Graphics Kongsberg AS';

	16#00000C5A:
		F_EtherCAT_VendorIDtoString := 'WOT Co.,Ltd.';

	16#00000C5C:
		F_EtherCAT_VendorIDtoString := 'SHENZHEN SENMUN ELECTRICAL CO.,LTD';

	16#00000C5D:
		F_EtherCAT_VendorIDtoString := 'Izhprest Ltd.';

	16#00000C5E:
		F_EtherCAT_VendorIDtoString := 'HAWE Hydraulik SE';

	16#00000C5F:
		F_EtherCAT_VendorIDtoString := 'Finetech GmbH & Co. KG';

	16#00000C60:
		F_EtherCAT_VendorIDtoString := 'Mitutoyo Corporation';

	16#00000C61:
		F_EtherCAT_VendorIDtoString := 'Cremer Speciaalmachines B.V.';

	16#00000C62:
		F_EtherCAT_VendorIDtoString := 'Astec Co., Ltd.';

	16#00000C64:
		F_EtherCAT_VendorIDtoString := 'ELNA LTD.';

	16#00000C65:
		F_EtherCAT_VendorIDtoString := 'Janasi Industries Ltd.';

	16#00000C66:
		F_EtherCAT_VendorIDtoString := 'Universidad de La Frontera, Facultad de Ingenieria y Ciencias, Centro de Modelacion y Computacion Cientifica (CEMCC)';

	16#00000C67:
		F_EtherCAT_VendorIDtoString := 'KALEJA GmbH';

	16#00000C68:
		F_EtherCAT_VendorIDtoString := 'Caldwell Machines & Tools trading as CMT Engineering';

	16#00000C69:
		F_EtherCAT_VendorIDtoString := 'ILJIN Global Holdings Co., Ltd.';

	16#00000C6A:
		F_EtherCAT_VendorIDtoString := 'Proteus Vietnam Limited';

	16#00000C6C:
		F_EtherCAT_VendorIDtoString := 'JUKI CORPORATION';

	16#00000C6D:
		F_EtherCAT_VendorIDtoString := 'MT Drive & Control (Shenzhen) Co.,Ltd';

	16#00000C6E:
		F_EtherCAT_VendorIDtoString := 'ShenZhen HongChuangXing Motion Technology Co.,Ltd';

	16#00000C6F:
		F_EtherCAT_VendorIDtoString := 'isMedia Co., Ltd.';

	16#00000C70:
		F_EtherCAT_VendorIDtoString := 'Shenzhen Yangshun Tongda Digital Technology Co., Ltd.';

	16#00000C71:
		F_EtherCAT_VendorIDtoString := 'MVTECH Co.,Ltd.';

	16#00000C72:
		F_EtherCAT_VendorIDtoString := 'Kane Terry Partridge dba Open Designer';

	16#00000C73:
		F_EtherCAT_VendorIDtoString := 'EK-Electronics GmbH';

	16#00000C74:
		F_EtherCAT_VendorIDtoString := 'Jiann Sheng Machinery & Electric Industrial Co., Ltd';

	16#00000C75:
		F_EtherCAT_VendorIDtoString := 'Gable Systems B.V.';

	16#00000C76:
		F_EtherCAT_VendorIDtoString := 'Constructions-3D SAS';

	16#00000C77:
		F_EtherCAT_VendorIDtoString := 'MIP robotics';

	16#00000C78:
		F_EtherCAT_VendorIDtoString := 'YouTool Automation Co., Ltd.';

	16#00000C79:
		F_EtherCAT_VendorIDtoString := 'Nanjing WEILAN Intelligent Technologies Co., Ltd.';

	16#00000C7A:
		F_EtherCAT_VendorIDtoString := 'ABB S.p.A.';

	16#00000C7B:
		F_EtherCAT_VendorIDtoString := 'Typhoon HIL Inc.';

	16#00000C7C:
		F_EtherCAT_VendorIDtoString := 'BLUTek Inc.';

	16#00000C7D:
		F_EtherCAT_VendorIDtoString := 'University of Engineering and Technology, Lahore, Al-Khwarizmi Institute of Computer Science, Human-Centered Robotics Lab';

	16#00000C7E:
		F_EtherCAT_VendorIDtoString := 'Technische Universitat Munchen, Fakultat fur Informatik, Lehrstuhl fur Robotik, Kunstliche Intelligenz und Echtzeitsysteme (Informatik 6)';

	16#00000C7F:
		F_EtherCAT_VendorIDtoString := 'Northrop Grumman Sperry Marine B.V. German Branch';

	16#00000C80:
		F_EtherCAT_VendorIDtoString := 'Technical University of Munich, Department of Electrical and Computer Engineering, Institute for Cognitive Systems (ICS)';

	16#00000C81:
		F_EtherCAT_VendorIDtoString := 'TNO';

	16#00000C82:
		F_EtherCAT_VendorIDtoString := 'IK Electronic Manufacturing Services S.L.U';

	16#00000C83:
		F_EtherCAT_VendorIDtoString := 'Ningbo Schleicher Technology Group Co., Ltd.';

	16#00000C84:
		F_EtherCAT_VendorIDtoString := 'TOWA Corporation';

	16#00000C85:
		F_EtherCAT_VendorIDtoString := 'Amacker Automation';

	16#00000C86:
		F_EtherCAT_VendorIDtoString := 'Hardt B.V.';

	16#00000C87:
		F_EtherCAT_VendorIDtoString := 'Anurichip System Inc.';

	16#00000C88:
		F_EtherCAT_VendorIDtoString := 'MESCO Engineering GmbH';

	16#00000C89:
		F_EtherCAT_VendorIDtoString := 'Oki Electric Industry Co., Ltd.';

	16#00000C8A:
		F_EtherCAT_VendorIDtoString := 'Motorsports Electronics, LLC';

	16#00000C8B:
		F_EtherCAT_VendorIDtoString := 'PPT Co., Ltd.';

	16#00000C8C:
		F_EtherCAT_VendorIDtoString := 'KYEONGIN TECH Co., Ltd.';

	16#00000C8D:
		F_EtherCAT_VendorIDtoString := 'SAS GYS';

	16#00000C8E:
		F_EtherCAT_VendorIDtoString := 'Cyber Surgery S.L.';

	16#00000C8F:
		F_EtherCAT_VendorIDtoString := 'CASTEK Mechatron Ind Co., Ltd.';

	16#00000C90:
		F_EtherCAT_VendorIDtoString := 'ERMAKSAN MAKINA SANAYI VE TICARET A.S.';

	16#00000C91:
		F_EtherCAT_VendorIDtoString := 'Elbit Systems Land Ltd.';

	16#00000C93:
		F_EtherCAT_VendorIDtoString := 'Javox Solutions GmbH';

	16#00000C94:
		F_EtherCAT_VendorIDtoString := 'Resilient Power Systems, Inc.';

	16#00000C95:
		F_EtherCAT_VendorIDtoString := 'CMRO Engineering';

	16#00000C96:
		F_EtherCAT_VendorIDtoString := 'Teknic, Inc.';

	16#00000C97:
		F_EtherCAT_VendorIDtoString := 'Lug Healthcare Technology S.L.';

	16#00000C98:
		F_EtherCAT_VendorIDtoString := 'Michael Koch GmbH';

	16#00000C99:
		F_EtherCAT_VendorIDtoString := 'UEC Scientific Instrument Co., Ltd.';

	16#00000C9A:
		F_EtherCAT_VendorIDtoString := 'WEISS GmbH';

	16#00000C9B:
		F_EtherCAT_VendorIDtoString := 'NITTOSEIKO CO., LTD.';

	16#00000C9C:
		F_EtherCAT_VendorIDtoString := 'WANTS Inc.';

	16#00000C9D:
		F_EtherCAT_VendorIDtoString := 'Tecnosens S.p.A.';

	16#00000C9F:
		F_EtherCAT_VendorIDtoString := 'Print Web International, Inc.';

	16#00000CA0:
		F_EtherCAT_VendorIDtoString := 'FAIR Innovation(Suzhou) Robot System Co.,Ltd.';

	16#00000CA1:
		F_EtherCAT_VendorIDtoString := 'OptiViz Technology, Inc.';

	16#00000CA2:
		F_EtherCAT_VendorIDtoString := 'Shanghai YISU Information Technologies Co.,Ltd.';

	16#00000CA3:
		F_EtherCAT_VendorIDtoString := 'Re S.p.A. Controlli Industriali';

	16#00000CA4:
		F_EtherCAT_VendorIDtoString := 'Canon Medical Systems Corporation';

	16#00000CA5:
		F_EtherCAT_VendorIDtoString := 'Suzhou Geyuan Electric Co., Ltd.';

	16#00000CA6:
		F_EtherCAT_VendorIDtoString := 'Shenzhen MICFIND Drive Technology Co., Ltd.';

	16#00000CA7:
		F_EtherCAT_VendorIDtoString := 'SECOM SRL';

	16#00000CA8:
		F_EtherCAT_VendorIDtoString := 'Panasonic Connect Co., Ltd.';

	16#00000CA9:
		F_EtherCAT_VendorIDtoString := 'BeiJing Agile Robots Technology Co.,Ltd.';

	16#00000CAB:
		F_EtherCAT_VendorIDtoString := 'Taiwan Innovative Space, Inc.';

	16#00000CAC:
		F_EtherCAT_VendorIDtoString := 'ABB Technikerschule';

	16#00000CAD:
		F_EtherCAT_VendorIDtoString := 'NOMOS Srl Tecnologie del Software';

	16#00000CAF:
		F_EtherCAT_VendorIDtoString := 'JSCC AUTOMATION (XIAMEN) LTD.';

	16#00000CB0:
		F_EtherCAT_VendorIDtoString := 'GMVT GmbH';

	16#00000CB1:
		F_EtherCAT_VendorIDtoString := 'Swisslog AG';

	16#00000CB2:
		F_EtherCAT_VendorIDtoString := 'Therm-x of California Inc.';

	16#00000CB3:
		F_EtherCAT_VendorIDtoString := 'CogniMade s.r.l.';

	16#00000CB4:
		F_EtherCAT_VendorIDtoString := 'SERT METAL SAS';

	16#00000CB5:
		F_EtherCAT_VendorIDtoString := 'Kardanan Shargh Co.';

	16#00000CB6:
		F_EtherCAT_VendorIDtoString := 'MPEX ROBOTICS KFT.';

	16#00000CB7:
		F_EtherCAT_VendorIDtoString := 'Critical Link LLC';

	16#00000CB8:
		F_EtherCAT_VendorIDtoString := 'Flokontrol Endustriyel Otomasyon San. ve Tic. Koll. Sti.';

	16#00000CB9:
		F_EtherCAT_VendorIDtoString := 'Nidec Avtron Automation Corporation';

	16#00000CBA:
		F_EtherCAT_VendorIDtoString := 'Alphasystem Co.,Ltd.';

	16#00000CBB:
		F_EtherCAT_VendorIDtoString := 'Carendes BVBA';

	16#00000CBC:
		F_EtherCAT_VendorIDtoString := 'Eltorque AS';

	16#00000CBD:
		F_EtherCAT_VendorIDtoString := 'University of Alberta, Faculty of Engineering';

	16#00000CBE:
		F_EtherCAT_VendorIDtoString := 'TOSIL Systems Private Limited';

	16#00000CBF:
		F_EtherCAT_VendorIDtoString := 'DELTA I/O CO.,LTD';

	16#00000CC0:
		F_EtherCAT_VendorIDtoString := 'Sipronika d.o.o.';

	16#00000CC1:
		F_EtherCAT_VendorIDtoString := 'TESA SARL';

	16#00000CC2:
		F_EtherCAT_VendorIDtoString := 'NXP B.V.';

	16#00000CC3:
		F_EtherCAT_VendorIDtoString := 'HERMOS AG';

	16#00000CC4:
		F_EtherCAT_VendorIDtoString := 'Svaya Robotics Pvt. Ltd.';

	16#00000CC5:
		F_EtherCAT_VendorIDtoString := 'ARRIVAL LTD.';

	16#00000CC6:
		F_EtherCAT_VendorIDtoString := 'Mold-Masters (2007) Limited';

	16#00000CC8:
		F_EtherCAT_VendorIDtoString := 'Hypex, d.o.o.';

	16#00000CC9:
		F_EtherCAT_VendorIDtoString := 'Sansei Technologies, Inc.';

	16#00000CCA:
		F_EtherCAT_VendorIDtoString := 'Shanghai United Imaging Healthcare Co., Ltd.';

	16#00000CCB:
		F_EtherCAT_VendorIDtoString := 'Seoul National University';

	16#00000CCC:
		F_EtherCAT_VendorIDtoString := '3C MACHINERY CO.,LTD.';

	16#00000CCD:
		F_EtherCAT_VendorIDtoString := 'CHINO CORPORATION';

	16#00000CCE:
		F_EtherCAT_VendorIDtoString := 'WUHAN MOTUS TECH CO.,LTD.';

	16#00000CCF:
		F_EtherCAT_VendorIDtoString := 'TPC Mechatronics Corp.';

	16#00000CD0:
		F_EtherCAT_VendorIDtoString := 'Philips Medical Systems DMC GmbH';

	16#00000CD1:
		F_EtherCAT_VendorIDtoString := 'TAZMO Co., Ltd.';

	16#00000CD2:
		F_EtherCAT_VendorIDtoString := 'Robo-Technology GmbH';

	16#00000CD3:
		F_EtherCAT_VendorIDtoString := 'Vivo Surgical Private Limited';

	16#00000CD4:
		F_EtherCAT_VendorIDtoString := 'Defence Research and Development Organisation, Research & Development Establishment (Engineers)';

	16#00000CD5:
		F_EtherCAT_VendorIDtoString := 'Jiangsu Shenzhou Semiconductor Technology Co., Ltd.';

	16#00000CD6:
		F_EtherCAT_VendorIDtoString := 'GrainSoft';

	16#00000CD7:
		F_EtherCAT_VendorIDtoString := 'MECCAD Sarl';

	16#00000CD9:
		F_EtherCAT_VendorIDtoString := 'National Formosa University, Department of Aeronautical Engineering, Innovative Design and Energy Application Lab. (IDEALab)';

	16#00000CDA:
		F_EtherCAT_VendorIDtoString := 'TOS Inc.';

	16#00000CDB:
		F_EtherCAT_VendorIDtoString := 'GTM Testing and Metrology GmbH';

	16#00000CDC:
		F_EtherCAT_VendorIDtoString := 'Prvni Signalni, a.s.';

	16#00000CDD:
		F_EtherCAT_VendorIDtoString := 'Georgia Institute of Technology, ECE Department, Center for Distributed Energy (CDE)';

	16#00000CDE:
		F_EtherCAT_VendorIDtoString := 'Plexim GmbH';

	16#00000CDF:
		F_EtherCAT_VendorIDtoString := 'Automation Industrial, Inc.';

	16#00000CE0:
		F_EtherCAT_VendorIDtoString := 'Regloplas AG';

	16#00000CE1:
		F_EtherCAT_VendorIDtoString := 'Azureus Solutions Ltd';

	16#00000CE2:
		F_EtherCAT_VendorIDtoString := 'Safran Electronics & Defense SAS';

	16#00000CE3:
		F_EtherCAT_VendorIDtoString := 'Sogeti Nederland B.V.';

	16#00000CE4:
		F_EtherCAT_VendorIDtoString := 'AKRYVIA SAS';

	16#00000CE5:
		F_EtherCAT_VendorIDtoString := 'FIRSTEC CO.,LTD.';

	16#00000CE6:
		F_EtherCAT_VendorIDtoString := 'M.D. Micro Detectors S.p.A.';

	16#00000CE7:
		F_EtherCAT_VendorIDtoString := 'Dataletics GmbH';

	16#00000CE8:
		F_EtherCAT_VendorIDtoString := 'Korea Institute of Machinery & Materials, Advanced Manufacturing Systems Research Division, Department of Ultra-Precision Machines and Systems';

	16#00000CE9:
		F_EtherCAT_VendorIDtoString := 'AEG Identifikationssysteme GmbH';

	16#00000CEA:
		F_EtherCAT_VendorIDtoString := 'CEA LIST';

	16#00000CEB:
		F_EtherCAT_VendorIDtoString := 'Shenyang Siasun Digital Drive Co., Ltd.';

	16#00000CEC:
		F_EtherCAT_VendorIDtoString := 'TissUse GmbH';

	16#00000CED:
		F_EtherCAT_VendorIDtoString := 'LithExx-Systems GmbH';

	16#00000CEE:
		F_EtherCAT_VendorIDtoString := 'AICRA s.r.o.';

	16#00000CEF:
		F_EtherCAT_VendorIDtoString := 'JANOME Corporation';

	16#00000CF0:
		F_EtherCAT_VendorIDtoString := 'Cambridge Filter Corporation';

	16#00000CF2:
		F_EtherCAT_VendorIDtoString := 'Celox Photonics Technology Inc.';

	16#00000CF3:
		F_EtherCAT_VendorIDtoString := 'swissQprint AG';

	16#00000CF4:
		F_EtherCAT_VendorIDtoString := 'COMFILE Technology INC.';

	16#00000CF5:
		F_EtherCAT_VendorIDtoString := 'Chengdu Vantron Technology Co., Ltd.';

	16#00000CF6:
		F_EtherCAT_VendorIDtoString := 'Duale Hochschule Baden-Wurttemberg Mannheim, Fakultat Technik, Studiengang Elektrotechnik';

	16#00000CF7:
		F_EtherCAT_VendorIDtoString := 'Tesollo Inc.';

	16#00000CF8:
		F_EtherCAT_VendorIDtoString := 'Roundpeg Technologies GmbH';

	16#00000CF9:
		F_EtherCAT_VendorIDtoString := 'Tianjin Research Institute of Electric Science Co.,Ltd.';

	16#00000CFB:
		F_EtherCAT_VendorIDtoString := 'Chicago Flyhouse, Inc.';

	16#00000CFC:
		F_EtherCAT_VendorIDtoString := 'Vectis Drive Inc.';

	16#00000CFD:
		F_EtherCAT_VendorIDtoString := 'IMSTec GmbH';

	16#00000CFE:
		F_EtherCAT_VendorIDtoString := 'Leibniz Universitat Hannover, Fakultat fur Elektrotechnik und Informatik, Institut fur Antriebssysteme und Leistungselektronik';

	16#00000CFF:
		F_EtherCAT_VendorIDtoString := 'Coretronic Corporation';

	16#00000D00:
		F_EtherCAT_VendorIDtoString := 'SOTHIS CIC TECH (Shanghai) Co., Ltd';

	16#00000D01:
		F_EtherCAT_VendorIDtoString := 'The Manufacturing Technology Centre Limited';

	16#00000D02:
		F_EtherCAT_VendorIDtoString := 'Tramper Technology B.V.';

	16#00000D03:
		F_EtherCAT_VendorIDtoString := 'Reaction Dynamics Lab Inc.';

	16#00000D04:
		F_EtherCAT_VendorIDtoString := 'Aeoon Technologies GmbH';

	16#00000D05:
		F_EtherCAT_VendorIDtoString := 'John Deere GmbH & Co. KG, John Deere Werk Mannheim';

	16#00000D06:
		F_EtherCAT_VendorIDtoString := 'Co.fin Elettronica s.r.l.';

	16#00000D07:
		F_EtherCAT_VendorIDtoString := 'CISWORKS GmbH & Co. KG';

	16#00000D09:
		F_EtherCAT_VendorIDtoString := 'Lucas-Nulle GmbH';

	16#00000D0A:
		F_EtherCAT_VendorIDtoString := 'Battelle Memorial Institute';

	16#00000D0B:
		F_EtherCAT_VendorIDtoString := 'Fine Logic Co., Ltd.';

	16#00000D0C:
		F_EtherCAT_VendorIDtoString := 'PACKR SAS';

	16#00000D0D:
		F_EtherCAT_VendorIDtoString := 'HP Indigo Ltd.';

	16#00000D0E:
		F_EtherCAT_VendorIDtoString := 'EMBEDDED SYSTEMS INC. dba ESI MOTION';

	16#00000D0F:
		F_EtherCAT_VendorIDtoString := 'DEIF A/S';

	16#00000D10:
		F_EtherCAT_VendorIDtoString := 'CEDRAT TECHNOLOGIES SA';

	16#00000D12:
		F_EtherCAT_VendorIDtoString := 'Givi Misure S.r.l. a socio unico';

	16#00000D13:
		F_EtherCAT_VendorIDtoString := 'ZETES Industries S.A.';

	16#00000D14:
		F_EtherCAT_VendorIDtoString := 'Ideaflex sp. z o.o.';

	16#00000D15:
		F_EtherCAT_VendorIDtoString := 'Emsiso d.o.o.';

	16#00000D16:
		F_EtherCAT_VendorIDtoString := 'SysTec Systemtechnik und Industrieautomation GmbH';

	16#00000D17:
		F_EtherCAT_VendorIDtoString := 'Soehnle Industrial Solutions GmbH';

	16#00000D18:
		F_EtherCAT_VendorIDtoString := 'Unizen Technologies Pvt. Ltd.';

	16#00000D19:
		F_EtherCAT_VendorIDtoString := 'White Oaks Engineering, LLC';

	16#00000D1A:
		F_EtherCAT_VendorIDtoString := 'Beijing BiTa Technical Services Co., Ltd.';

	16#00000D1B:
		F_EtherCAT_VendorIDtoString := 'Nordmann GmbH & Co. KG';

	16#00000D1C:
		F_EtherCAT_VendorIDtoString := 'Seven Metal Corp.';

	16#00000D1D:
		F_EtherCAT_VendorIDtoString := 'Festo Korea Co., Ltd.';

	16#00000D1E:
		F_EtherCAT_VendorIDtoString := 'Hyperspectral Sciences, Inc.';

	16#00000D1F:
		F_EtherCAT_VendorIDtoString := 'AA EDM Corporation';

	16#00000D20:
		F_EtherCAT_VendorIDtoString := 'Corelase Oy';

	16#00000D21:
		F_EtherCAT_VendorIDtoString := 'CETHIK Group Co., Ltd';

	16#00000D22:
		F_EtherCAT_VendorIDtoString := 'LIVSMED, Inc.';

	16#00000D23:
		F_EtherCAT_VendorIDtoString := 'Hochschule Munchen';

	16#00000D24:
		F_EtherCAT_VendorIDtoString := 'WSA:Automation';

	16#00000D26:
		F_EtherCAT_VendorIDtoString := 'Universitat Stuttgart, Fakultat Konstruktions-, Produktions- und Fahrzeugtechnik, Institut fur Systemdynamik';

	16#00000D27:
		F_EtherCAT_VendorIDtoString := 'AXIOS 3D Services GmbH';

	16#00000D28:
		F_EtherCAT_VendorIDtoString := 'CASCINATION AG';

	16#00000D29:
		F_EtherCAT_VendorIDtoString := 'Kontinent ETS LLC';

	16#00000D2B:
		F_EtherCAT_VendorIDtoString := 'STXI Motion Ltd.';

	16#00000D2C:
		F_EtherCAT_VendorIDtoString := 'RFHIC Corporation';

	16#00000D2D:
		F_EtherCAT_VendorIDtoString := 'Technische Universitat Wien, Fakultat fur Maschinenwesen und Betriebswissenschaften, Institut fur Fertigungstechnik und Photonische Technologien';

	16#00000D2E:
		F_EtherCAT_VendorIDtoString := 'RT Corporation';

	16#00000D2F:
		F_EtherCAT_VendorIDtoString := 'Automation Controls Group, a Division of Milwaukee Electronics Corporation';

	16#00000D30:
		F_EtherCAT_VendorIDtoString := 'AIRS Medical Inc.';

	16#00000D31:
		F_EtherCAT_VendorIDtoString := 'Cardinal Scale Manufacturing Company';

	16#00000D32:
		F_EtherCAT_VendorIDtoString := 'Mehta Cad Cam Systems Pvt. Ltd.';

	16#00000D33:
		F_EtherCAT_VendorIDtoString := 'TWERD Power Electronics';

	16#00000D34:
		F_EtherCAT_VendorIDtoString := 'Canon Nanotechnologies Inc.';

	16#00000D35:
		F_EtherCAT_VendorIDtoString := 'Karlsruher Institut fur Technologie, Fakultat fur Elektrotechnik und Informationstechnik, Institut fur Elektroenergiesysteme und Hochspannungstechnik';

	16#00000D36:
		F_EtherCAT_VendorIDtoString := 'Beijing Grand Hitek Co., Ltd.';

	16#00000D37:
		F_EtherCAT_VendorIDtoString := 'Soft Control (Shenzhen) Automation Technology Co., Ltd';

	16#00000D38:
		F_EtherCAT_VendorIDtoString := 'Y2 Corporation';

	16#00000D39:
		F_EtherCAT_VendorIDtoString := 'Posts and Telecommunications Institute of Technology, Ho Chi Minh City (PTIT-HCM), Electronics 2 Department, Automatic Control Division';

	16#00000D3A:
		F_EtherCAT_VendorIDtoString := 'RoPeM Solution Co., Ltd.';

	16#00000D3B:
		F_EtherCAT_VendorIDtoString := 'SEPION TECHNOLOGY INC.';

	16#00000D3C:
		F_EtherCAT_VendorIDtoString := 'TRUMPF Lasersystems for Semiconductor Manufacturing AG';

	16#00000D3D:
		F_EtherCAT_VendorIDtoString := 'Sagentia Limited';

	16#00000D3F:
		F_EtherCAT_VendorIDtoString := 'ColorPartner GmbH';

	16#00000D40:
		F_EtherCAT_VendorIDtoString := 'Dongguan embedfire Electronic Technology Co., Ltd.';

	16#00000D41:
		F_EtherCAT_VendorIDtoString := 'Cell-Vit Co., Ltd.';

	16#00000D42:
		F_EtherCAT_VendorIDtoString := 'East China University of Science and Technology, School of Chemistry and Molecular Engineering, Nanopore Single Molecule Detection Laboratory';

	16#00000D43:
		F_EtherCAT_VendorIDtoString := 'Vanwyk Systems B.V.';

	16#00000D44:
		F_EtherCAT_VendorIDtoString := 'NGK INSULATORS, LTD.';

	16#00000D45:
		F_EtherCAT_VendorIDtoString := 'NIHON KOSHUHA Co., Ltd.';

	16#00000D46:
		F_EtherCAT_VendorIDtoString := 'HEMERIA SAS';

	16#00000D47:
		F_EtherCAT_VendorIDtoString := 'Qmax Systems India Pvt. Ltd.';

	16#00000D48:
		F_EtherCAT_VendorIDtoString := 'TENDLY ENTERPRISES CO., LTD.';

	16#00000D49:
		F_EtherCAT_VendorIDtoString := 'Chenghuan Technology (Shenzhen) Co., Ltd.';

	16#00000D4A:
		F_EtherCAT_VendorIDtoString := 'Shanghai Weihong Automation Technology Co., Ltd.';

	16#00000D4B:
		F_EtherCAT_VendorIDtoString := 'Uster Technologies (China) Co., Ltd.';

	16#00000D4C:
		F_EtherCAT_VendorIDtoString := 'MGI Tech Co., Ltd.';

	16#00000D4D:
		F_EtherCAT_VendorIDtoString := 'KELI MOTOR GROUP CO., LTD.';

	16#00000D4E:
		F_EtherCAT_VendorIDtoString := 'Carlo Gavazzi Ltd. (Malta)';

	16#00000D50:
		F_EtherCAT_VendorIDtoString := 'Optiflux NV';

	16#00000D51:
		F_EtherCAT_VendorIDtoString := 'Mistral Solutions Pvt. Ltd.';

	16#00000D52:
		F_EtherCAT_VendorIDtoString := 'Fraunhofer-Institut fur Windenergiesysteme IWES';

	16#00000D53:
		F_EtherCAT_VendorIDtoString := 'Enekom Enerji Bilisim ve Muhendislik San Tic A.S.';

	16#00000D54:
		F_EtherCAT_VendorIDtoString := 'MASEP Medical Science & Technology Development (Shenzhen) Co., Ltd.';

	16#00000D55:
		F_EtherCAT_VendorIDtoString := 'Shenzhen Soogeen Electronics Co., LTD.';

	16#00000D56:
		F_EtherCAT_VendorIDtoString := 'UJin Technology, Inc.';

	16#00000D57:
		F_EtherCAT_VendorIDtoString := 'TOSEI SYSTEMS CO., LTD.';

	16#00000D58:
		F_EtherCAT_VendorIDtoString := 'TAIYO, LTD.';

	16#00000D59:
		F_EtherCAT_VendorIDtoString := 'Alloc Corporation';

	16#00000D5A:
		F_EtherCAT_VendorIDtoString := 'WaferPath, Inc.';

	16#00000D5B:
		F_EtherCAT_VendorIDtoString := 'Genesis Dimensions LLC';

	16#00000D5C:
		F_EtherCAT_VendorIDtoString := 'Zhuhai Tai-Action Electronics Co., Ltd.';

	16#00000D5D:
		F_EtherCAT_VendorIDtoString := 'JSC Diakont';

	16#00000D5E:
		F_EtherCAT_VendorIDtoString := 'SCHNEKON Automation (Shanghai) Co.,Ltd.';

	16#00000D5F:
		F_EtherCAT_VendorIDtoString := 'NSI-MI Technologies LLC';

	16#00000D60:
		F_EtherCAT_VendorIDtoString := 'JD Squared, Inc.';

	16#00000D61:
		F_EtherCAT_VendorIDtoString := 'Sanctuary Cognitive Systems Corporation';

	16#00000D62:
		F_EtherCAT_VendorIDtoString := 'NICEMACH CO., LTD.';

	16#00000D63:
		F_EtherCAT_VendorIDtoString := 'ERTURK MAKINE SAN TIC. LTD. STI';

	16#00000D64:
		F_EtherCAT_VendorIDtoString := 'Surgnova Healthcare Technologies (Beijing) Co., Ltd.';

	16#00000D65:
		F_EtherCAT_VendorIDtoString := 'soniKKs Ultrasonics Technology GmbH';

	16#00000D66:
		F_EtherCAT_VendorIDtoString := 'NBB Controls + Components GmbH';

	16#00000D68:
		F_EtherCAT_VendorIDtoString := 'OOO "NPP Mera"';

	16#00000D69:
		F_EtherCAT_VendorIDtoString := 'Poulten Selfe & Lee Ltd';

	16#00000D6A:
		F_EtherCAT_VendorIDtoString := 'Monolithic Power Systems, Inc.';

	16#00000D6B:
		F_EtherCAT_VendorIDtoString := 'UK Atomic Energy Authority, RACE';

	16#00000D6C:
		F_EtherCAT_VendorIDtoString := 'PULS GmbH';

	16#00000D6D:
		F_EtherCAT_VendorIDtoString := 'FUGEN CO., LTD';

	16#00000D6E:
		F_EtherCAT_VendorIDtoString := 'coboworx GmbH';

	16#00000D6F:
		F_EtherCAT_VendorIDtoString := 'A&D Company, Limited';

	16#00000D70:
		F_EtherCAT_VendorIDtoString := 'JOOWON TECHNOLOGY Co., Ltd.';

	16#00000D71:
		F_EtherCAT_VendorIDtoString := 'ODC Co., Ltd.';

	16#00000D72:
		F_EtherCAT_VendorIDtoString := 'Asyril SA';

	16#00000D73:
		F_EtherCAT_VendorIDtoString := 'Robotics Robotics (Shenzhen) Ltd.';

	16#00000D74:
		F_EtherCAT_VendorIDtoString := 'Automated Precision Inc.';

	16#00000D75:
		F_EtherCAT_VendorIDtoString := 'Ozyegin University, Faculty of Engineering, Department of Mechanical Engineering, Robotics Laboratory';

	16#00000D76:
		F_EtherCAT_VendorIDtoString := 'Fujikura Ltd.';

	16#00000D77:
		F_EtherCAT_VendorIDtoString := 'Relativity Space, Inc.';

	16#00000D78:
		F_EtherCAT_VendorIDtoString := 'Hangzhou Core Control Robotics CO.,LTD';

	16#00000D79:
		F_EtherCAT_VendorIDtoString := 'Beijing Shangcon Intelligent Technology Co., Ltd.';

	16#00000D7A:
		F_EtherCAT_VendorIDtoString := 'Panasonic Advanced Technology Development Co.,Ltd.';

	16#00000D7B:
		F_EtherCAT_VendorIDtoString := 'Philips Electronics Nederland B.V. Philips Engineering Solutions';

	16#00000D7C:
		F_EtherCAT_VendorIDtoString := 'Emoco Labs AB';

	16#00000D7D:
		F_EtherCAT_VendorIDtoString := 'Otto Heuss GmbH';

	16#00000D7F:
		F_EtherCAT_VendorIDtoString := 'PRAUCON';

	16#00000D80:
		F_EtherCAT_VendorIDtoString := 'Ashby Microsystems Ltd';

	16#00000D81:
		F_EtherCAT_VendorIDtoString := 'Suzhou Veichi Electric Co., Ltd';

	16#00000D82:
		F_EtherCAT_VendorIDtoString := 'SCAME SISTEMI S.R.L.';

	16#00000D83:
		F_EtherCAT_VendorIDtoString := 'J.M. Voith SE & Co KG';

	16#00000D84:
		F_EtherCAT_VendorIDtoString := 'Sier Motor (Dongguan) Co., Ltd.';

	16#00000D85:
		F_EtherCAT_VendorIDtoString := 'Shanghai Wingbow Precision Technology Co.,Ltd.';

	16#00000D86:
		F_EtherCAT_VendorIDtoString := 'Mertech Elektronik Arge Sanayi ve Ticaret Anonim Sirketi';

	16#00000D87:
		F_EtherCAT_VendorIDtoString := 'Summa nv';

	16#00000D88:
		F_EtherCAT_VendorIDtoString := 'Bucher Hydraulics AG Frutigen';

	16#00000D89:
		F_EtherCAT_VendorIDtoString := 'Pulse Structural Monitoring Ltd';

	16#00000D8A:
		F_EtherCAT_VendorIDtoString := 'Sanovo Technology Netherlands B.V.';

	16#00000D8B:
		F_EtherCAT_VendorIDtoString := 'ACCRETECH POWERTRO SYSTEM CO., LTD.';

	16#00000D8C:
		F_EtherCAT_VendorIDtoString := 'TOYOTA INDUSTRIES CORPORATION';

	16#00000D8D:
		F_EtherCAT_VendorIDtoString := 'KOEM CO., LTD.';

	16#00000D8E:
		F_EtherCAT_VendorIDtoString := 'Beijing NAURA Microelectronics Equipment Co., Ltd.';

	16#00000D8F:
		F_EtherCAT_VendorIDtoString := 'NEXT Prototypes e.V.';

	16#00000D90:
		F_EtherCAT_VendorIDtoString := 'Ningbo Advance Automation Technology Co.,Ltd.';

	16#00000D91:
		F_EtherCAT_VendorIDtoString := 'TRUMPF Laser SE';

	16#00000D92:
		F_EtherCAT_VendorIDtoString := 'Asensus Surgical, Inc.';

	16#00000D93:
		F_EtherCAT_VendorIDtoString := 'Exluce Inc.';

	16#00000D94:
		F_EtherCAT_VendorIDtoString := 'Computer Gesteuerte Systeme GmbH';

	16#00000D95:
		F_EtherCAT_VendorIDtoString := 'ALSTOM Belgium SA';

	16#00000D96:
		F_EtherCAT_VendorIDtoString := 'HG-Tronik';

	16#00000D97:
		F_EtherCAT_VendorIDtoString := 'HAFNER Pneumatika Kft.';

	16#00000D98:
		F_EtherCAT_VendorIDtoString := 'Intigia S.L.';

	16#00000D99:
		F_EtherCAT_VendorIDtoString := 'Next Generation Rail Technologies S.L.';

	16#00000D9A:
		F_EtherCAT_VendorIDtoString := 'APEX Semiconductors (USA) Co., Ltd.';

	16#00000D9B:
		F_EtherCAT_VendorIDtoString := 'True Velocity Ammunition, LLC';

	16#00000D9C:
		F_EtherCAT_VendorIDtoString := 'Anderson Electric Controls, Inc.';

	16#00000D9E:
		F_EtherCAT_VendorIDtoString := 'Exonetik Inc.';

	16#00000D9F:
		F_EtherCAT_VendorIDtoString := 'R&D Test Systems A/S';

	16#00000DA0:
		F_EtherCAT_VendorIDtoString := 'SDP (Shanghai) Industrial Corporation Ltd.';

	16#00000DA1:
		F_EtherCAT_VendorIDtoString := 'NOVASEN Co., Ltd.';

	16#00000DA2:
		F_EtherCAT_VendorIDtoString := 'RTDS Technologies Inc.';

	16#00000DA3:
		F_EtherCAT_VendorIDtoString := 'CPI Vertex Antennentechnik GmbH';

	16#00000DA4:
		F_EtherCAT_VendorIDtoString := 'Eindhoven Medical Robotics B.V.';

	16#00000DA5:
		F_EtherCAT_VendorIDtoString := 'QEI Corporation';

	16#00000DA6:
		F_EtherCAT_VendorIDtoString := 'Reliste Ges.m.b.H.';

	16#00000DA7:
		F_EtherCAT_VendorIDtoString := 'ABL Space Systems';

	16#00000DA8:
		F_EtherCAT_VendorIDtoString := 'PostProcess Technologies, Inc.';

	16#00000DA9:
		F_EtherCAT_VendorIDtoString := 'SEcontrol Automation (Shanghai) Co., Ltd.';

	16#00000DAA:
		F_EtherCAT_VendorIDtoString := 'Phoenix Contact Asia-Pacific (Nanjing) Co., Ltd.';

	16#00000DAB:
		F_EtherCAT_VendorIDtoString := 'Heal Force Huayao Biological Technology (Shanghai) Co., Ltd';

	16#00000DAC:
		F_EtherCAT_VendorIDtoString := 'Spellman High Voltage Electronics Ltd.';

	16#00000DAD:
		F_EtherCAT_VendorIDtoString := 'Wipro GE Healthcare Private Limited';

	16#00000DAE:
		F_EtherCAT_VendorIDtoString := 'KOFLOC Corp.';

	16#00000DAF:
		F_EtherCAT_VendorIDtoString := 'Niryo SAS';

	16#00000DB0:
		F_EtherCAT_VendorIDtoString := 'Friedrich Maschinen- und Werkzeugbau GmbH';

	16#00000DB1:
		F_EtherCAT_VendorIDtoString := 'Togatec Sarl';

	16#00000DB2:
		F_EtherCAT_VendorIDtoString := 'EDAG Engineering GmbH';

	16#00000DB3:
		F_EtherCAT_VendorIDtoString := 'Arius Technology Inc.';

	16#00000DB4:
		F_EtherCAT_VendorIDtoString := 'ROKKO SYSTEMS PTE LTD';

	16#00000DB5:
		F_EtherCAT_VendorIDtoString := 'Novotechnik Messwertaufnehmer OHG';

	16#00000DB6:
		F_EtherCAT_VendorIDtoString := 'Shanghai Chenzhu Instrument Co.,LTD';

	16#00000DB7:
		F_EtherCAT_VendorIDtoString := 'Yantai Free Intelligent Equipment Co.,Ltd.';

	16#00000DB8:
		F_EtherCAT_VendorIDtoString := 'The University of Newcastle, College of Engineering Science and Environment, School of Engineering';

	16#00000DB9:
		F_EtherCAT_VendorIDtoString := 'California Polytechnic State University, College of Engineering, Computer Engineering Department';

	16#00000DBA:
		F_EtherCAT_VendorIDtoString := 'PRACTEK Technology Co., Ltd.';

	16#00000DBC:
		F_EtherCAT_VendorIDtoString := 'Ningbo Longtai Medical Technology Co., Ltd.';

	16#00000DBD:
		F_EtherCAT_VendorIDtoString := 'Fulling & Partner Ingenieurgesellschaft mbH';

	16#00000DBE:
		F_EtherCAT_VendorIDtoString := 'TechMagic, Inc.';

	16#00000DBF:
		F_EtherCAT_VendorIDtoString := 'Bagtech International Pty Ltd';

	16#00000DC0:
		F_EtherCAT_VendorIDtoString := 'DCO Systems Ltd';

	16#00000DC1:
		F_EtherCAT_VendorIDtoString := 'Shenzhen Pengxing Intelligence Research Co., Ltd.';

	16#00000DC2:
		F_EtherCAT_VendorIDtoString := 'Sunny Instruments Singapore Pte Ltd';

	16#00000DC3:
		F_EtherCAT_VendorIDtoString := 'Tokyo Denki University, School of Science and Technology for Future Life, Department of Robotics and Mechatronics';

	16#00000DC4:
		F_EtherCAT_VendorIDtoString := 'RMD Engineering Inc.';

	16#00000DC5:
		F_EtherCAT_VendorIDtoString := 'Ganzhou Zhongke TOYODA Intelligent Equipment Technology Co., Ltd.';

	16#00000DC6:
		F_EtherCAT_VendorIDtoString := 'Feurer Automation AG';

	16#00000DC7:
		F_EtherCAT_VendorIDtoString := 'Surpass Industry Co., Ltd.';

	16#00000DC8:
		F_EtherCAT_VendorIDtoString := 'PLC2 Design GmbH';

	16#00000DC9:
		F_EtherCAT_VendorIDtoString := 'Elesa S.p.A.';

	16#00000DCA:
		F_EtherCAT_VendorIDtoString := 'SHENYANG KING CAREER TECHNOLOGY CO.,LTD.';

	16#00000DCB:
		F_EtherCAT_VendorIDtoString := 'NexCOBOT Taiwan Co., Ltd.';

	16#00000DCC:
		F_EtherCAT_VendorIDtoString := 'HOERBIGER Flow Control GmbH';

	16#00000DCD:
		F_EtherCAT_VendorIDtoString := 'Karl Dungs GmbH & Co. KG';

	16#00000DCE:
		F_EtherCAT_VendorIDtoString := 'KRONO-SAFE, SAS';

	16#00000DCF:
		F_EtherCAT_VendorIDtoString := 'Merz Maschinenfabrik GmbH';

	16#00000DD0:
		F_EtherCAT_VendorIDtoString := 'EKS InTec GmbH';

	16#00000DD1:
		F_EtherCAT_VendorIDtoString := 'HiSilicon (Shanghai) Technologies Co., Ltd.';

	16#00000DD2:
		F_EtherCAT_VendorIDtoString := 'Jiangsu JITRI Sioux Technologies Co.,Ltd.';

	16#00000DD3:
		F_EtherCAT_VendorIDtoString := 'ConTeK, spol. s.r.o.';

	16#00000DD4:
		F_EtherCAT_VendorIDtoString := 'Dr. Hubert GmbH';

	16#00000DD5:
		F_EtherCAT_VendorIDtoString := 'DELTATEC s.a.';

	16#00000DD6:
		F_EtherCAT_VendorIDtoString := 'ShangHai LeiTong Technology Center Co., Ltd.';

	16#00000DD7:
		F_EtherCAT_VendorIDtoString := 'Shanghai Xinrui Drive Technology Co., Ltd.';

	16#00000DD8:
		F_EtherCAT_VendorIDtoString := 'Macnica Galaxy International Limited';

	16#00000DDA:
		F_EtherCAT_VendorIDtoString := 'PICODE Corp.';

	16#00000DDB:
		F_EtherCAT_VendorIDtoString := 'VGD Engineering Ltd.';

	16#00000DDC:
		F_EtherCAT_VendorIDtoString := 'WIRobotics Inc.';

	16#00000DDD:
		F_EtherCAT_VendorIDtoString := 'Xingyu Electron (NINGBO) Co.,Ltd.';

	16#00000DDE:
		F_EtherCAT_VendorIDtoString := 'Yamaki Electric Corporation';

	16#00000DDF:
		F_EtherCAT_VendorIDtoString := 'MST Co., Ltd.';

	16#00000DE0:
		F_EtherCAT_VendorIDtoString := 'Brinkmann Electronic Berlin GmbH';

	16#00000DE1:
		F_EtherCAT_VendorIDtoString := 'Mazor Robotics Ltd.';

	16#00000DE2:
		F_EtherCAT_VendorIDtoString := 'Center for Power Electronics and Drives';

	16#00000DE3:
		F_EtherCAT_VendorIDtoString := 'SINTEF Energi AS';

	16#00000DE4:
		F_EtherCAT_VendorIDtoString := 'Suzhou ST-Intelligence Technology Co., Ltd.';

	16#00000DE5:
		F_EtherCAT_VendorIDtoString := 'GEFASOFT Automatisierung und Software GmbH Regensburg';

	16#00000DE6:
		F_EtherCAT_VendorIDtoString := 'Shenzhen AS-AI Technology Co., Ltd.';

	16#00000DE7:
		F_EtherCAT_VendorIDtoString := 'Shenzhen Beilai Technology Co.,Ltd';

	16#00000DE8:
		F_EtherCAT_VendorIDtoString := 'PETER HIRT GmbH';

	16#00000DE9:
		F_EtherCAT_VendorIDtoString := 'ADTEC Technology Inc.';

	16#00000DEA:
		F_EtherCAT_VendorIDtoString := 'SEMICS Inc.';

	16#00000DEB:
		F_EtherCAT_VendorIDtoString := 'Digitronik Labs Inc.';

	16#00000DEC:
		F_EtherCAT_VendorIDtoString := 'University of Denver, Ritchie School of Engineering and Computer Science, Department of Mechanical and Materials Engineering, Robotics, Locomotion, and Control Lab';

	16#00000DED:
		F_EtherCAT_VendorIDtoString := 'Capto UG (haftungsbeschrankt)';

	16#00000DEE:
		F_EtherCAT_VendorIDtoString := 'DST Draxlmaier Systemtechnik GmbH';

	16#00000DEF:
		F_EtherCAT_VendorIDtoString := 'Rototest International AB';

	16#00000DF0:
		F_EtherCAT_VendorIDtoString := 'Shenzhen DH-Robotics Technology Co.,Ltd.';

	16#00000DF1:
		F_EtherCAT_VendorIDtoString := 'Centre Suisse dElectronique et de Microtechnique';

	16#00000DF2:
		F_EtherCAT_VendorIDtoString := 'DIGALOG Industrie-Mikroelektronik GmbH';

	16#00000DF3:
		F_EtherCAT_VendorIDtoString := 'Gevasol Feedback Technologies Ltd.';

	16#00000DF4:
		F_EtherCAT_VendorIDtoString := 'Jiangsu Gtake Electric Co., Ltd.';

	16#00000DF5:
		F_EtherCAT_VendorIDtoString := 'Thermo Fisher Scientific Inc.';

	16#00000DF6:
		F_EtherCAT_VendorIDtoString := 'Stony MicroWorks LTD';

	16#00000DF8:
		F_EtherCAT_VendorIDtoString := 'Shanghai Tayor Heavy Industry(Group) Co., Ltd.';

	16#00000DF9:
		F_EtherCAT_VendorIDtoString := 'Heartland.Data Inc.';

	16#00000DFA:
		F_EtherCAT_VendorIDtoString := 'FLSmidth Pfister GmbH';

	16#00000DFB:
		F_EtherCAT_VendorIDtoString := 'Viscom AG';

	16#00000DFC:
		F_EtherCAT_VendorIDtoString := 'Toyo Label Co., Ltd.';

	16#00000DFD:
		F_EtherCAT_VendorIDtoString := 'Harbin Sagebot Intelligent Medical Equipment Co., Ltd.';

	16#00000DFE:
		F_EtherCAT_VendorIDtoString := 'TGA Industries Limited';

	16#00000E00:
		F_EtherCAT_VendorIDtoString := 'Phase 1 Engineering, LLC';

	16#00000E01:
		F_EtherCAT_VendorIDtoString := 'EGON HARIG GmbH';

	16#00000E02:
		F_EtherCAT_VendorIDtoString := 'I.A.S.G. Kereskedelmi es Szolgaltato Kft.';

	16#00000E03:
		F_EtherCAT_VendorIDtoString := 'MONS University, Faculty of Engineering, Department of Electromagnetism and Telecommunications';

	16#00000E04:
		F_EtherCAT_VendorIDtoString := 'Technische Universitat Munchen, TUM School of Engineering and Design, Lehrstuhl fur Produktentwicklung und Leichtbau';

	16#00000E05:
		F_EtherCAT_VendorIDtoString := 'eCential Robotics';

	16#00000E06:
		F_EtherCAT_VendorIDtoString := 'D.Electron S.r.l.';

	16#00000E08:
		F_EtherCAT_VendorIDtoString := 'Shenzhen CSL Vacuum Science And Technology Co., Ltd.';

	16#00000E09:
		F_EtherCAT_VendorIDtoString := 'Guangdong Tiantai Robot Co., Ltd.';

	16#00000E0A:
		F_EtherCAT_VendorIDtoString := 'Delta Networks (Xiamen) LTD.';

	16#00000E0B:
		F_EtherCAT_VendorIDtoString := 'Ignitarium Technology Solutions Private Limited';

	16#00000E0C:
		F_EtherCAT_VendorIDtoString := 'Graco Inc.';

	16#00000E0D:
		F_EtherCAT_VendorIDtoString := 'Shenyang Guangcheng Technology Co., Ltd.';

	16#00000E0E:
		F_EtherCAT_VendorIDtoString := 'Dongguan Xunwei Intelligent Technology  Co., Ltd.';

	16#00000E0F:
		F_EtherCAT_VendorIDtoString := 'Schubert Elektroanlagen GmbH';

	16#00000E10:
		F_EtherCAT_VendorIDtoString := 'Ruian CITIC Electronic Equipment Co., Ltd.';

	16#00000E11:
		F_EtherCAT_VendorIDtoString := 'DynaMotion GmbH';

	16#00000E12:
		F_EtherCAT_VendorIDtoString := 'Inxpect S.p.A.';

	16#00000E14:
		F_EtherCAT_VendorIDtoString := 'Shenzhen Sincevision Technology Co., Ltd';

	16#00000E15:
		F_EtherCAT_VendorIDtoString := 'LMT Lichtmesstechnik GmbH Berlin';

	16#00000E16:
		F_EtherCAT_VendorIDtoString := 'DAWONSYS Co., Ltd.';

	16#00000E17:
		F_EtherCAT_VendorIDtoString := 'Guangzhou JKE Automation Equipment Co., Ltd.';

	16#00000E18:
		F_EtherCAT_VendorIDtoString := 'ASBISc Enterprises PLC';

	16#00000E19:
		F_EtherCAT_VendorIDtoString := 'University of Pennsylvania, School of Arts & Sciences, Department of Physics & Astronomy';

	16#00000E1A:
		F_EtherCAT_VendorIDtoString := 'electronics-lis';

	16#00000E1B:
		F_EtherCAT_VendorIDtoString := 'Otto Zimmermann GmbH';

	16#00000E1C:
		F_EtherCAT_VendorIDtoString := 'Schneider Electric Asia Pte Ltd';

	16#00000E1D:
		F_EtherCAT_VendorIDtoString := 'Shenzhen Matribox Intelligent Technology Co.,Ltd.';

	16#00000E1E:
		F_EtherCAT_VendorIDtoString := 'UnitX, Inc.';

	16#00000E1F:
		F_EtherCAT_VendorIDtoString := 'Bitrode Corporation';

	16#00000E20:
		F_EtherCAT_VendorIDtoString := 'NL Automation';

	16#00000E21:
		F_EtherCAT_VendorIDtoString := 'ORing (Shanghai) Corp.';

	16#00000E22:
		F_EtherCAT_VendorIDtoString := 'JuHeng Aero Systems Technology Co., Ltd.';

	16#00000E23:
		F_EtherCAT_VendorIDtoString := 'Addverb Technologies Limited';

	16#00000E24:
		F_EtherCAT_VendorIDtoString := 'HiFuture S.r.l.';

	16#00000E25:
		F_EtherCAT_VendorIDtoString := 'Kuwana Metals Finetech, Ltd.';

	16#00000E27:
		F_EtherCAT_VendorIDtoString := 'MinMaxMedical SAS';

	16#00000E28:
		F_EtherCAT_VendorIDtoString := 'Weifang Lokomo Precision Industry Co., Ltd.';

	16#00000E29:
		F_EtherCAT_VendorIDtoString := 'MegaChips Corporation';

	16#00000E2A:
		F_EtherCAT_VendorIDtoString := 'University of Debrecen, Faculty of Engineering, Department of Mechatronics';

	16#00000E2B:
		F_EtherCAT_VendorIDtoString := 'Quarry Electron Design, LLC';

	16#00000E2C:
		F_EtherCAT_VendorIDtoString := 'Spellman High Voltage Electronics Corporation';

	16#00000E2D:
		F_EtherCAT_VendorIDtoString := 'Offshore Renewable Energy Catapult Ltd.';

	16#00000E2E:
		F_EtherCAT_VendorIDtoString := 'Shenzhen Noke Technology Co., Ltd.';

	16#00000E2F:
		F_EtherCAT_VendorIDtoString := 'Shanghai MRDcom Co., Ltd.';

	16#00000E30:
		F_EtherCAT_VendorIDtoString := 'National Applied Research Laboratories, Taiwan Instrument Research Institute';

	16#00000E31:
		F_EtherCAT_VendorIDtoString := 'Psicontrol N.V.';

	16#00000E32:
		F_EtherCAT_VendorIDtoString := 'Eugenus, Inc.';

	16#00000E33:
		F_EtherCAT_VendorIDtoString := 'Shenzhen Ligent Sensor Tech Co., Ltd.';

	16#00000E34:
		F_EtherCAT_VendorIDtoString := 'South-Central Minzu University, College of Computer Science';

	16#00000E35:
		F_EtherCAT_VendorIDtoString := 'Shanghai Tekgao Information & Technology Co.,Ltd';

	16#00000E36:
		F_EtherCAT_VendorIDtoString := 'Beijing Dahao Technology Corp.,Ltd';

	16#00000E37:
		F_EtherCAT_VendorIDtoString := 'Nanjing Lanhao Intelligent Technology Co., Ltd.';

	16#00000E38:
		F_EtherCAT_VendorIDtoString := 'Heiberger Solutions Inc';

	16#00000E39:
		F_EtherCAT_VendorIDtoString := 'Thinkwintek Co., Ltd.';

	16#00000E3B:
		F_EtherCAT_VendorIDtoString := 'Novity Inc';

	16#00000E3C:
		F_EtherCAT_VendorIDtoString := 'ADM Automation Ltd.';

	16#00000E3D:
		F_EtherCAT_VendorIDtoString := 'Fortress Interlocks Limited';

	16#00000E3E:
		F_EtherCAT_VendorIDtoString := 'Ningbo AirTAC Automatic Industrial Co., Ltd.';

	16#00000E3F:
		F_EtherCAT_VendorIDtoString := 'Shanghai SODRON Automatic Co., Ltd.';

	16#00000E40:
		F_EtherCAT_VendorIDtoString := 'Sichuan Injet Electric Co., Ltd.';

	16#00000E41:
		F_EtherCAT_VendorIDtoString := 'Zumbach Electronic AG';

	16#00000E42:
		F_EtherCAT_VendorIDtoString := 'Cohu GmbH';

	16#00000E43:
		F_EtherCAT_VendorIDtoString := 'Ilitron Enerji ve Bilgi Teknolojileri A.Ş.';

	16#00000E44:
		F_EtherCAT_VendorIDtoString := '&Hunan Staim Microelectronics Co., Ltd.';

	16#00000E45:
		F_EtherCAT_VendorIDtoString := 'ADTEC Plasma Technology Korea Co., Ltd.';

	16#00000E46:
		F_EtherCAT_VendorIDtoString := 'BAADER Food Systems Denmark A/S';

	16#00000E47:
		F_EtherCAT_VendorIDtoString := 'Koh Young Technology Inc.';

	16#00000E48:
		F_EtherCAT_VendorIDtoString := 'Balem Co., Ltd.';

	16#00000E49:
		F_EtherCAT_VendorIDtoString := 'Fidus Systems Inc.';

	16#00000E4A:
		F_EtherCAT_VendorIDtoString := 'Isabellenhutte Heusler GmbH & Co. KG';

	16#00000E4C:
		F_EtherCAT_VendorIDtoString := 'Huazhong University of Science & Technology (HUST), School of Mechanical Science & Engineering';

	16#00000E4D:
		F_EtherCAT_VendorIDtoString := 'Suzhou Servo Dynamics Co.,Ltd.';

	16#00000E4E:
		F_EtherCAT_VendorIDtoString := 'Nanchang Slater Automation System Co., Ltd.';

	16#00000E4F:
		F_EtherCAT_VendorIDtoString := 'Pixsys Srl';

	16#00000E50:
		F_EtherCAT_VendorIDtoString := 'DTS INSIGHT Corporation';

	16#00000E51:
		F_EtherCAT_VendorIDtoString := 'Leijenaar Electronics';

	16#00000E52:
		F_EtherCAT_VendorIDtoString := 'Zhejiang TaiBangXingPu intelligent science&technology co., ltd.';

	16#00000E53:
		F_EtherCAT_VendorIDtoString := 'Sunrise Instruments Co.,Ltd.';

	16#00000E54:
		F_EtherCAT_VendorIDtoString := 'Microtest S.r.l.';

	16#00000E55:
		F_EtherCAT_VendorIDtoString := 'Xinhe (Beijing) Data Technology Co., Ltd.';

	16#00000E56:
		F_EtherCAT_VendorIDtoString := 'Anzo Controls Private Limited';

	16#00000E57:
		F_EtherCAT_VendorIDtoString := 'Guangzhou Jinglun Automation Equipment Co., Ltd.';

	16#00000E58:
		F_EtherCAT_VendorIDtoString := 'TG-Packaging BV';

	16#00000E59:
		F_EtherCAT_VendorIDtoString := 'Hefei Weichong Technology Co., Ltd.';

	16#00000E5A:
		F_EtherCAT_VendorIDtoString := 'Cyrola Inc.';

	16#00000E5C:
		F_EtherCAT_VendorIDtoString := 'SDMC America Technology Inc.';

	16#00000E5D:
		F_EtherCAT_VendorIDtoString := 'Convergent RnR Ltd.';

	16#00000E5E:
		F_EtherCAT_VendorIDtoString := 'EV Group E. Thallner GmbH';

	16#00000E5F:
		F_EtherCAT_VendorIDtoString := 'Medtronic, Inc.';

	16#00000E60:
		F_EtherCAT_VendorIDtoString := 'Nautilus Systems, Inc.';

	16#00000E62:
		F_EtherCAT_VendorIDtoString := 'Wack Engineering';

	16#00000E63:
		F_EtherCAT_VendorIDtoString := 'Luminous Show Technology Limited';

	16#00000E64:
		F_EtherCAT_VendorIDtoString := 'Dexmart Technology Corp.';

	16#00000E65:
		F_EtherCAT_VendorIDtoString := 'Prevas A/S';

	16#00000E66:
		F_EtherCAT_VendorIDtoString := 'Funcience Corporation';

	16#00000E67:
		F_EtherCAT_VendorIDtoString := 'H. ZANDER GmbH & Co. KG';

	16#00000E68:
		F_EtherCAT_VendorIDtoString := 'Fasford Technology Co., Ltd.';

	16#00000E69:
		F_EtherCAT_VendorIDtoString := 'Agito Akribis Systems Ltd.';

	16#00000E6A:
		F_EtherCAT_VendorIDtoString := 'Alberts NV';

	16#00000E6B:
		F_EtherCAT_VendorIDtoString := 'LINX Corporation';

	16#00000E6C:
		F_EtherCAT_VendorIDtoString := 'Wuxi Silicon Field Microelectronics Co.,Ltd.';

	16#00000E6D:
		F_EtherCAT_VendorIDtoString := 'General Fusion Inc.';

	16#00000E6E:
		F_EtherCAT_VendorIDtoString := 'InfoSocket Co., Ltd.';

	16#00000E6F:
		F_EtherCAT_VendorIDtoString := 'Honda R&D Co., Ltd.';

	16#00000E70:
		F_EtherCAT_VendorIDtoString := 'Renesas Electronics India Private Limited';

	16#00000E71:
		F_EtherCAT_VendorIDtoString := 'NOVO Engineering, Inc.';

	16#00000E72:
		F_EtherCAT_VendorIDtoString := 'TIANJIN SEAGULLROBOT AUTOMATION TECHNOLOGY LIMITED';

	16#00000E73:
		F_EtherCAT_VendorIDtoString := 'Mogensen GmbH & Co. KG';

	16#00000E74:
		F_EtherCAT_VendorIDtoString := 'Strategy Enabled Solutions, LLC';

	16#00000E75:
		F_EtherCAT_VendorIDtoString := 'AKC Angersbach + Kaiser Computer GmbH';

	16#00000E76:
		F_EtherCAT_VendorIDtoString := 'HIWIN Technologies Corp.';

	16#00000E77:
		F_EtherCAT_VendorIDtoString := 'Rex Bionics Ltd';

	16#00000E78:
		F_EtherCAT_VendorIDtoString := 'FACTS Engineering, LLC';

	16#00000E79:
		F_EtherCAT_VendorIDtoString := 'CI SYSTEMS (ISRAEL) LTD.';

	16#00000E7A:
		F_EtherCAT_VendorIDtoString := 'Momentis Surgical Ltd.';

	16#00000E7B:
		F_EtherCAT_VendorIDtoString := 'Origin Co., Ltd.';

	16#00000E7C:
		F_EtherCAT_VendorIDtoString := 'Shandong ITLC Electric Technology Co.,Ltd';

	16#00000E7D:
		F_EtherCAT_VendorIDtoString := 'Vebu Labs, Inc';

	16#00000E7E:
		F_EtherCAT_VendorIDtoString := 'KCF Technologies, Inc.';

	16#00000E7F:
		F_EtherCAT_VendorIDtoString := 'Aalto University, School of Science, Department of Neuroscience and Biomedical Engineering, TMS Group';

	16#00000E80:
		F_EtherCAT_VendorIDtoString := 'Jiangsu Gaokai Precision Fluid Technology Co., Ltd.';

	16#00000E82:
		F_EtherCAT_VendorIDtoString := 'Shanghai Lanbao Sensing Technology Co., Ltd.';

	16#00000E83:
		F_EtherCAT_VendorIDtoString := 'Guangdong Tianji Robot Co., Ltd.';

	16#00000E84:
		F_EtherCAT_VendorIDtoString := 'Beijing Aibo Mechanics & Electrics Co., Ltd';

	16#00000E85:
		F_EtherCAT_VendorIDtoString := 'Shanghai Yinguan Semiconductor Technology Co., Ltd.';

	16#00000E86:
		F_EtherCAT_VendorIDtoString := 'Wuhan Gewei Electronic Technologies Co., Ltd.';

	16#00000E87:
		F_EtherCAT_VendorIDtoString := 'ALTAM Systems SL';

	16#00000E88:
		F_EtherCAT_VendorIDtoString := 'Four Technos Co., Ltd.';

	16#00000E89:
		F_EtherCAT_VendorIDtoString := 'Midea Welling Motor Technology (Shanghai) Co., Ltd.';

	16#00000E8B:
		F_EtherCAT_VendorIDtoString := 'NINGBO DEGSON TECHNOLOGY CO., LTD';

	16#00000E8C:
		F_EtherCAT_VendorIDtoString := 'YANTAI DERON INDUSTRY CO.,LTD';

	16#00000E8D:
		F_EtherCAT_VendorIDtoString := '3Sigma SARL';

	16#00000E8E:
		F_EtherCAT_VendorIDtoString := 'Rethink Robotics GmbH';

	16#00000E8F:
		F_EtherCAT_VendorIDtoString := 'Auroma Technologies Co., LLC DBA Access Laser Company';

	16#00000E90:
		F_EtherCAT_VendorIDtoString := 'JIANGSU LIHE I&C TECHNOLOGY CO., LTD.';

	16#00000E91:
		F_EtherCAT_VendorIDtoString := 'HangZhou TongHang Edrive Technology Co.,Ltd.';

	16#00000E92:
		F_EtherCAT_VendorIDtoString := 'Hangzhou DAREN Technology CO.,LTD.';

	16#00000E93:
		F_EtherCAT_VendorIDtoString := 'Orbotech Ltd.';

	16#00000E94:
		F_EtherCAT_VendorIDtoString := 'Feejoy Technology (Shanghai) Co., Ltd.';

	16#00000E95:
		F_EtherCAT_VendorIDtoString := 'Xiamen Yudian Automation Technology Co., Ltd.';

	16#00000E96:
		F_EtherCAT_VendorIDtoString := 'Shenzhen Chuanneng Automation Co., Ltd.';

	16#00000E97:
		F_EtherCAT_VendorIDtoString := 'Southern University of Science and Technology, College of Engineering, Department of Mechanical and Energy Engineering';

	16#00000E98:
		F_EtherCAT_VendorIDtoString := 'Honda Electronics Co., Ltd.';

	16#00000E99:
		F_EtherCAT_VendorIDtoString := 'Ningbo Anson CNC Technique Co., Ltd';

	16#00000E9A:
		F_EtherCAT_VendorIDtoString := 'Shenzhen Akusense Technology Co., Ltd.';

	16#00000E9B:
		F_EtherCAT_VendorIDtoString := 'Systemtechnik LEBER GmbH & Co. KG';

	16#00000E9C:
		F_EtherCAT_VendorIDtoString := 'SERVOneering GmbH';

	16#00000E9E:
		F_EtherCAT_VendorIDtoString := 'Optotune Switzerland AG';

	16#00000E9F:
		F_EtherCAT_VendorIDtoString := 'Precision Sensors Division of United Electric Controls';

	16#00000EA0:
		F_EtherCAT_VendorIDtoString := 'University of Arkansas, College of Engineering, Department of Electrical Engineering';

	16#00000EA1:
		F_EtherCAT_VendorIDtoString := 'SHINKAWA Sensor Technology, Inc.';

	16#00000EA2:
		F_EtherCAT_VendorIDtoString := 'Continental Automotive Technologies GmbH';

	16#00000EA3:
		F_EtherCAT_VendorIDtoString := 'Changzhou Kunwei Sensing Technology Co.,Ltd.';

	16#00000EA5:
		F_EtherCAT_VendorIDtoString := 'Shanghai Huayuan Chuangxin Software Co., Ltd.';

	16#00000EA6:
		F_EtherCAT_VendorIDtoString := 'C-ENSYS';

	16#00000EA7:
		F_EtherCAT_VendorIDtoString := 'Terma Technologies GmbH';

	16#00000EA8:
		F_EtherCAT_VendorIDtoString := 'Hangzhou J-Drv Servo Technology Co., Ltd.';

	16#00000EA9:
		F_EtherCAT_VendorIDtoString := 'FononTech B.V.';

	16#00000EAA:
		F_EtherCAT_VendorIDtoString := 'AI-GmbH-KVU';

	16#00000EAB:
		F_EtherCAT_VendorIDtoString := 'SAS STC';

	16#00000EAC:
		F_EtherCAT_VendorIDtoString := 'Sygnal Technologies, Inc.';

	16#00000EAD:
		F_EtherCAT_VendorIDtoString := 'PSTEK Co., Ltd';

	16#00000EAE:
		F_EtherCAT_VendorIDtoString := 'Shanghai Huatai Digital Control Co., Ltd.';

	16#00000EAF:
		F_EtherCAT_VendorIDtoString := 'Startingames SAS';

	16#00000EB0:
		F_EtherCAT_VendorIDtoString := 'Guangzhou Aosong Electronic Co., Ltd.';

	16#00000EB1:
		F_EtherCAT_VendorIDtoString := 'Yantai Aitron Robotic Technology Co., Ltd.';

	16#00000EB3:
		F_EtherCAT_VendorIDtoString := 'QSD Sistemi srl';

	16#00000EB4:
		F_EtherCAT_VendorIDtoString := 'TDK-Lambda Corporation';

	16#00000EB5:
		F_EtherCAT_VendorIDtoString := 'Advanced Electronic Designs, Inc.';

	16#00000EB6:
		F_EtherCAT_VendorIDtoString := 'PLIEM (Shanghai) Intelligent Technology Co., Ltd.';

	16#00000EB7:
		F_EtherCAT_VendorIDtoString := 'Everfoton Technologies Corporation Limited';

	16#00000EB8:
		F_EtherCAT_VendorIDtoString := 'KARL STORZ VentureONE Germany GmbH';

	16#00000EB9:
		F_EtherCAT_VendorIDtoString := 'Cove Technology Consulting LLC';

	16#00000EBA:
		F_EtherCAT_VendorIDtoString := 'Noah Medical Inc';

	16#00000EBB:
		F_EtherCAT_VendorIDtoString := 'Philips Health Technology (China) Co., Ltd. Shenyang Branch';

	16#00000EBC:
		F_EtherCAT_VendorIDtoString := 'Shanghai Flexem Technology Co.,Ltd.';

	16#00000EBD:
		F_EtherCAT_VendorIDtoString := 'Xiamen Codefair Semiconductor Technology Co., Ltd.';

	16#00000EBE:
		F_EtherCAT_VendorIDtoString := 'Maschinenfabrik Reinhausen GmbH';

	16#00000EBF:
		F_EtherCAT_VendorIDtoString := 'Automationdirect.com Inc.';

	16#00000EC0:
		F_EtherCAT_VendorIDtoString := 'Rheinmetall Air Defence AG';

	16#00000EC1:
		F_EtherCAT_VendorIDtoString := 'El Camino GmbH Training - Engineering - Consultancy';

	16#00000EC2:
		F_EtherCAT_VendorIDtoString := 'Mohawk International Services BV';

	16#00000EC3:
		F_EtherCAT_VendorIDtoString := 'MELTIN MMI Co., Ltd.';

	16#00000EC4:
		F_EtherCAT_VendorIDtoString := 'JBG-Elektronik GmbH';

	16#00000EC5:
		F_EtherCAT_VendorIDtoString := 'E.C.S. Sistemi Elettronici S.p.A';

	16#00000EC6:
		F_EtherCAT_VendorIDtoString := 'ForceN Inc.';

	16#00000EC7:
		F_EtherCAT_VendorIDtoString := 'REELEX Packaging Solutions, Inc.';

	16#00000EC8:
		F_EtherCAT_VendorIDtoString := 'CUBICON Inc.';

	16#00000EC9:
		F_EtherCAT_VendorIDtoString := 'Hyosung Corporation';

	16#00000ECA:
		F_EtherCAT_VendorIDtoString := 'IGS Inc.';

	16#00000ECB:
		F_EtherCAT_VendorIDtoString := 'Beijing Jingyi Automation Equipment Co., Ltd.';

	16#00000ECC:
		F_EtherCAT_VendorIDtoString := 'Aitalmac (Nanjing) Stonework And Mechanical Co.,LTD.';

	16#00000ECD:
		F_EtherCAT_VendorIDtoString := 'Durr Systems AG';

	16#00000ECE:
		F_EtherCAT_VendorIDtoString := 'POUNDFUL ELECTRONICS CO., LTD.';

	16#00000ECF:
		F_EtherCAT_VendorIDtoString := 'Kuka Robotics Guangdong Co., Ltd.';

	16#00000ED0:
		F_EtherCAT_VendorIDtoString := 'Kratos Analytical Ltd';

	16#00000ED1:
		F_EtherCAT_VendorIDtoString := 'Fortive Setra-ICG (Tianjin) Co., Ltd.';

	16#00000ED3:
		F_EtherCAT_VendorIDtoString := 'Speedgoat GmbH';

	16#00000ED4:
		F_EtherCAT_VendorIDtoString := 'Airbus Defence and Space S.A.U.';

	16#00000ED5:
		F_EtherCAT_VendorIDtoString := 'W Endoluminal Robotics Ltd.';

	16#00000ED6:
		F_EtherCAT_VendorIDtoString := 'II-VI Aerospace & Defense, Inc.';

	16#00000ED7:
		F_EtherCAT_VendorIDtoString := 'Shenzhen SZD Technology Co., Ltd.';

	16#00000ED8:
		F_EtherCAT_VendorIDtoString := 'Electrical Engineering Institute Nikola Tesla Joint Stock Company Belgrade';

	16#00000ED9:
		F_EtherCAT_VendorIDtoString := 'FRECON Electric (Shenzhen) Co., Ltd.';

	16#00000EDA:
		F_EtherCAT_VendorIDtoString := 'Acevin Solutions';

	16#00000EDB:
		F_EtherCAT_VendorIDtoString := 'EDB Srl';

	16#00000EDC:
		F_EtherCAT_VendorIDtoString := 'Bosch Global Software Technologies Private Limited';

	16#00000EDD:
		F_EtherCAT_VendorIDtoString := 'ABB E-mobility B.V.';

	16#00000EDE:
		F_EtherCAT_VendorIDtoString := 'EUMAX (Shanghai) Corp.';

	16#00000EDF:
		F_EtherCAT_VendorIDtoString := 'Mitsui Electron Co., Ltd.';

	16#00000EE0:
		F_EtherCAT_VendorIDtoString := 'ForSight Robotics Ltd.';

	16#00000EE1:
		F_EtherCAT_VendorIDtoString := 'ICON Technology, Inc.';

	16#00000EE2:
		F_EtherCAT_VendorIDtoString := 'Amitech Electronics Design';

	16#00000EE3:
		F_EtherCAT_VendorIDtoString := 'Renesas Design Vietnam Co., Ltd.';

	16#00000EE4:
		F_EtherCAT_VendorIDtoString := 'AMESS Co.,Ltd.';

	16#00000EE5:
		F_EtherCAT_VendorIDtoString := 'Hexar s.r.l.';

	16#00000EE6:
		F_EtherCAT_VendorIDtoString := 'Shenzhen Lewo Electric Technology Co., Ltd.';

	16#00000EE7:
		F_EtherCAT_VendorIDtoString := 'Vrije Universiteit Brussel, Faculty of Engineering, Department of Mechanical Engineering';

	16#00000EE8:
		F_EtherCAT_VendorIDtoString := '1MRobotics LTD';

	16#00000EE9:
		F_EtherCAT_VendorIDtoString := 'Baumer Innovation GmbH';

	16#00000EEA:
		F_EtherCAT_VendorIDtoString := 'Fargo Engineering, Inc.';

	16#00000EEB:
		F_EtherCAT_VendorIDtoString := 'Tesla Inc.';

	16#00000EED:
		F_EtherCAT_VendorIDtoString := 'Eagle Wing Design';

	16#00000EEE:
		F_EtherCAT_VendorIDtoString := 'Espotel Oy';

	16#00000EEF:
		F_EtherCAT_VendorIDtoString := 'Guangzhou Chenkong Intelligent Technology Co., Ltd.';

	16#00000EF0:
		F_EtherCAT_VendorIDtoString := 'Elite Robots Co., Ltd.';

	16#00000EF1:
		F_EtherCAT_VendorIDtoString := 'STORK IMM B.V.';

	16#00000EF2:
		F_EtherCAT_VendorIDtoString := 'Rheinmetall Soldier Electronics GmbH';

	16#00000EF4:
		F_EtherCAT_VendorIDtoString := 'ELARABY-Toyoichi Engineering Corporation';

	16#00000EF5:
		F_EtherCAT_VendorIDtoString := 'WISDRI (Wuhan) Automation Co., Ltd.';

	16#00000EF6:
		F_EtherCAT_VendorIDtoString := 'Koutechs Co., Ltd.';

	16#00000EF7:
		F_EtherCAT_VendorIDtoString := 'TECNA S.p.A.';

	16#00000EF8:
		F_EtherCAT_VendorIDtoString := 'TAMS Firmware Co., Ltd.';

	16#00000EF9:
		F_EtherCAT_VendorIDtoString := 'Lenovo (Shanghai) Information Technology Co., Ltd.';

	16#00000EFA:
		F_EtherCAT_VendorIDtoString := 'Foshan Zhiang Technology Co., Ltd.';

	16#00000EFB:
		F_EtherCAT_VendorIDtoString := 'Lachmann & Rink GmbH';

	16#00000EFC:
		F_EtherCAT_VendorIDtoString := 'Daifuku Co., Ltd.';

	16#00000EFE:
		F_EtherCAT_VendorIDtoString := 'Sodick Co., Ltd.';

	16#00000EFF:
		F_EtherCAT_VendorIDtoString := 'FUZHOU FU CHANG WECON ELECTRONIC TECHNOLOGY CO., LTD';

	16#00000F00:
		F_EtherCAT_VendorIDtoString := 'Zhongke Times (Shenzhen) Computer System Co., Ltd.';

	16#00000F01:
		F_EtherCAT_VendorIDtoString := 'New Scale Technologies, Inc.';

	16#00000F02:
		F_EtherCAT_VendorIDtoString := 'GCLAB MUHENDİSLİK A.Ş.';

	16#00000F03:
		F_EtherCAT_VendorIDtoString := 'BERNSTEIN AG';

	16#00000F04:
		F_EtherCAT_VendorIDtoString := 'Malvern Panalytical B.V.';

	16#00000F05:
		F_EtherCAT_VendorIDtoString := 'University of Illinois Urbana-Champaign, The Granger College of Engineering, Control Systems Laboratory';

	16#00000F06:
		F_EtherCAT_VendorIDtoString := 'Suzhou Bogute Intelligent Manufacturing Co., Ltd.';

	16#00000F07:
		F_EtherCAT_VendorIDtoString := 'Guangdong Anda Automation Solutions Co., Ltd.';

	16#00000F08:
		F_EtherCAT_VendorIDtoString := 'Shenzhen Rspower Technology Co., Ltd.';

	16#00000F09:
		F_EtherCAT_VendorIDtoString := 'Twenty Three BV';

	16#00000F0A:
		F_EtherCAT_VendorIDtoString := 'Tec Gihan Co., Ltd.';

	16#00000F0B:
		F_EtherCAT_VendorIDtoString := 'Distalmotion SA';

	16#00000F0C:
		F_EtherCAT_VendorIDtoString := 'HAPTION SA';

	16#00000F0E:
		F_EtherCAT_VendorIDtoString := 'Zimmer GmbH';

	16#00000F0F:
		F_EtherCAT_VendorIDtoString := 'Neuralink Corporation';

	16#00000F10:
		F_EtherCAT_VendorIDtoString := 'AUXIND S.r.l.';

	16#00000F11:
		F_EtherCAT_VendorIDtoString := 'Sony Group Corporation';

	16#00000F12:
		F_EtherCAT_VendorIDtoString := 'Eletrica Ballmann Ltda';

	16#00000F13:
		F_EtherCAT_VendorIDtoString := 'Jiangsu Fenghesheng Intelligent Technology Co., Ltd.';

	16#00000F14:
		F_EtherCAT_VendorIDtoString := 'Fujian Speciband Technology Co., Ltd.';

	16#00000F15:
		F_EtherCAT_VendorIDtoString := 'Hyleecon (Qingdao) Technology Co.,Ltd.';

	16#00000F16:
		F_EtherCAT_VendorIDtoString := 'Xiamen Kudom Electronic Technology Co., Ltd';

	16#00000F17:
		F_EtherCAT_VendorIDtoString := 'Wuhan Fingu Electronic Technology Co., Ltd.';

	16#00000F19:
		F_EtherCAT_VendorIDtoString := 'DELO Industrie Klebstoffe GmbH & Co. KGaA';

	16#00000F1A:
		F_EtherCAT_VendorIDtoString := 'FIAtec GmbH';

	16#00000F1B:
		F_EtherCAT_VendorIDtoString := 'Hiteco S.r.l.';

	16#00000F1C:
		F_EtherCAT_VendorIDtoString := 'DMS Co., Ltd.';

	16#00000F1D:
		F_EtherCAT_VendorIDtoString := 'Shandong Shanke Intelligent Control Digital Technology Co., Ltd';

	16#00000F1E:
		F_EtherCAT_VendorIDtoString := 'NanJing iNVOEE Technology CO.,LTD';

	16#00000F1F:
		F_EtherCAT_VendorIDtoString := 'BEx-Solution GmbH';

	16#00000F20:
		F_EtherCAT_VendorIDtoString := 'Second Order Effects, Inc';

	16#00000F21:
		F_EtherCAT_VendorIDtoString := 'SALZ Automation GmbH';

	16#00000F22:
		F_EtherCAT_VendorIDtoString := 'Couth Infotech Private Limited';

	16#00000F23:
		F_EtherCAT_VendorIDtoString := 'Avnet Electronics Technology (China) Limited';

	16#00000F24:
		F_EtherCAT_VendorIDtoString := 'Malvern Panalytical Limited';

	16#00000F26:
		F_EtherCAT_VendorIDtoString := 'Polygon T.R Ltd.';

	16#00000F28:
		F_EtherCAT_VendorIDtoString := 'MysteryCrafters LLC';

	16#00000F29:
		F_EtherCAT_VendorIDtoString := 'Benezan Electronics';

	16#00000F2A:
		F_EtherCAT_VendorIDtoString := 'Rockist Automation technology (suzhou) Co., LTD';

	16#00000F2B:
		F_EtherCAT_VendorIDtoString := 'Hangzhou Kuntai Maglev Technology Co., Ltd.';

	16#00000F2C:
		F_EtherCAT_VendorIDtoString := 'SCADA d.o.o';

	16#00000F2D:
		F_EtherCAT_VendorIDtoString := 'CHANGZHOU JKONGMOTOR CO., LTD';

	16#00000F2E:
		F_EtherCAT_VendorIDtoString := 'Erhardt+Leimer GmbH';

	16#00000F2F:
		F_EtherCAT_VendorIDtoString := 'Acinotech (RF) Pty Ltd';

	16#00000F30:
		F_EtherCAT_VendorIDtoString := 'Beijing Cotytech Co.,LTD.';

	16#00000F31:
		F_EtherCAT_VendorIDtoString := 'Danfoss Technologies Pvt. Ltd.';

	16#00000F32:
		F_EtherCAT_VendorIDtoString := 'Beijing Baihui Weikang Technology Co., Ltd.';

	16#00000F33:
		F_EtherCAT_VendorIDtoString := 'University of York, School of Physics, Engineering and Technology, Intelligent Hybrid Robotics Lab';

	16#00000F34:
		F_EtherCAT_VendorIDtoString := 'Beijing Dotouch Information Technology Co., Ltd.';

	16#00000F35:
		F_EtherCAT_VendorIDtoString := 'Centre for Development of Advanced Computing, Power Electronics Group';

	16#00000F36:
		F_EtherCAT_VendorIDtoString := 'Moog Industrial Control (Suzhou) Co., Ltd.';

	16#00000F37:
		F_EtherCAT_VendorIDtoString := 'HUNAN LINGXIAN MAGLEV TECHNOLOGY CO. LTD';

	16#00000F38:
		F_EtherCAT_VendorIDtoString := 'FB Project S.R.L.';

	16#00000F39:
		F_EtherCAT_VendorIDtoString := 'Ionautics AB';

	16#00000F3A:
		F_EtherCAT_VendorIDtoString := 'Helion Energy, Inc.';

	16#00000F3B:
		F_EtherCAT_VendorIDtoString := 'OND Co., Ltd.';

	16#00000F3C:
		F_EtherCAT_VendorIDtoString := 'Sysmetric Ltd.';

	16#00000F3D:
		F_EtherCAT_VendorIDtoString := 'Shenzhen Safetop Tech Co., Ltd.';

	16#00000F3E:
		F_EtherCAT_VendorIDtoString := 'FZI Forschungszentrum Informatik';

	16#00000F3F:
		F_EtherCAT_VendorIDtoString := 'Pollen Robotics SAS';

	16#00000F40:
		F_EtherCAT_VendorIDtoString := 'Colombian Imaging Technologies S.A.S';

	16#00000F41:
		F_EtherCAT_VendorIDtoString := 'Sollae Systems Co., Ltd.';

	16#00000F42:
		F_EtherCAT_VendorIDtoString := 'MP bvba (CTRL engineering)';

	16#00000F43:
		F_EtherCAT_VendorIDtoString := 'DAgostino Industries Group, Inc.';

	16#00000F44:
		F_EtherCAT_VendorIDtoString := 'Akrodyn GmbH';

	16#00000F45:
		F_EtherCAT_VendorIDtoString := 'Continental Automation Systems Pvt Ltd';

	16#00000F46:
		F_EtherCAT_VendorIDtoString := 'CRRC QINGDAO SIFANG CO.,LTD.';

	16#00000F47:
		F_EtherCAT_VendorIDtoString := 'JST Inc.';

	16#00000F48:
		F_EtherCAT_VendorIDtoString := 'magniX USA, Inc';

	16#00000F49:
		F_EtherCAT_VendorIDtoString := 'Shenzhen ForYou Technology Co., Ltd.';

	16#00000F4A:
		F_EtherCAT_VendorIDtoString := 'Hebei Bode Tech Technology Co., Ltd.';

	16#00000F4B:
		F_EtherCAT_VendorIDtoString := 'ISRA VISION GmbH';

	16#00000F4C:
		F_EtherCAT_VendorIDtoString := 'Indian Institute of Science, Centre for Product Design and Manufacturing';

	16#00000F4D:
		F_EtherCAT_VendorIDtoString := 'PT. WEQ TECHNOLOGI INDONESIA';

	16#00000F4E:
		F_EtherCAT_VendorIDtoString := 'Precitec Optronik GmbH';

	16#00000F4F:
		F_EtherCAT_VendorIDtoString := 'EURL MICROPROCESSOR';

	16#00000F50:
		F_EtherCAT_VendorIDtoString := 'NIHO-MOTORS Export-Import d.o.o. Konjic';

	16#00000F51:
		F_EtherCAT_VendorIDtoString := 'Przedsiębiorstwo Usług Elektronicznych TRAK sp.j.';

	16#00000F52:
		F_EtherCAT_VendorIDtoString := 'dosmatix GmbH';

	16#00000F53:
		F_EtherCAT_VendorIDtoString := 'WPG China (SZ) Inc.';

	16#00000F55:
		F_EtherCAT_VendorIDtoString := 'Animotech Inc.';

	16#00000F56:
		F_EtherCAT_VendorIDtoString := 'Vertigo Designs LLC';

	16#00000F57:
		F_EtherCAT_VendorIDtoString := 'Suzhou Shenen Electronic Technology Co.,Ltd.';

	16#00000F58:
		F_EtherCAT_VendorIDtoString := 'EC Engineering Korea Co.,Ltd.';

	16#00000F59:
		F_EtherCAT_VendorIDtoString := 'Artinchip Technology Co., Ltd.';

	16#00000F5A:
		F_EtherCAT_VendorIDtoString := 'OSAIcnc S.r.l.';

	16#00000F5B:
		F_EtherCAT_VendorIDtoString := 'Multiscan Technologies SL';

	16#00000F5C:
		F_EtherCAT_VendorIDtoString := 'DIGITAL CONTROL S.R.L.';

	16#00000F5D:
		F_EtherCAT_VendorIDtoString := 'MARS Optoelectronica S.R.L.';

	16#00000F5E:
		F_EtherCAT_VendorIDtoString := 'AURA Inc., NOIRLab';

	16#00000F5F:
		F_EtherCAT_VendorIDtoString := 'Xiamen Wain Electrical Co., Ltd.';

	16#00000F60:
		F_EtherCAT_VendorIDtoString := 'Shanghai B&A Automation System Co.,Ltd';

	16#00000F61:
		F_EtherCAT_VendorIDtoString := 'Controlway (Suzhou) Electric Co., Ltd.';

	16#00000F62:
		F_EtherCAT_VendorIDtoString := 'FORMOSA PLASTICS CORPORATION';

	16#00000F63:
		F_EtherCAT_VendorIDtoString := 'Soluware GmbH';

	16#00000F64:
		F_EtherCAT_VendorIDtoString := 'Sonic Italia S.r.l.';

	16#00000F65:
		F_EtherCAT_VendorIDtoString := 'WireFlow AB';

	16#00000F66:
		F_EtherCAT_VendorIDtoString := 'MeetFuture Technology (Shanghai) Co., Ltd.';

	16#00000F67:
		F_EtherCAT_VendorIDtoString := 'Pentamaster Instrumentation Sdn. Bhd.';

	16#00000F68:
		F_EtherCAT_VendorIDtoString := 'Shenzhen Xiaobai Automation Technology Co., Ltd.';

	16#00000F69:
		F_EtherCAT_VendorIDtoString := 'Acorn Logic Technology Corp.';

	16#00000F6A:
		F_EtherCAT_VendorIDtoString := 'Dankook University, College of Engineering, School of Electronics and Electrical Engineering, Dankook University Power Electronics Laboratory (DUPEL)';

	16#00000F6B:
		F_EtherCAT_VendorIDtoString := 'PACKAGING TECHNOLOGIES & INSPECTION, LLC';

	16#00000F6C:
		F_EtherCAT_VendorIDtoString := 'iMAR Navigation GmbH';

	16#00000F6D:
		F_EtherCAT_VendorIDtoString := 'ISP Co., Ltd.';

	16#00000F6E:
		F_EtherCAT_VendorIDtoString := 'Telsys LTD';

	16#00000F6F:
		F_EtherCAT_VendorIDtoString := 'Brandenburgische Technische Universitat Cottbus-Senftenberg, Fakultat 3 Maschinenbau, Elektro- und Energiesysteme, Institut fur Elektrische und Thermische Energiesysteme, Lehrstuhl Leistungselektronik und Antriebssysteme';

	16#00000F70:
		F_EtherCAT_VendorIDtoString := 'Primetals Technologies Germany GmbH';

	16#00000F71:
		F_EtherCAT_VendorIDtoString := 'JAY Electronique S.A.S.';

	16#00000F72:
		F_EtherCAT_VendorIDtoString := 'KBM Automation AG';

	16#00000F73:
		F_EtherCAT_VendorIDtoString := 'STEP SCIENCE CO., LTD.';

	16#00000F74:
		F_EtherCAT_VendorIDtoString := 'Amazon.com Services LLC';

	16#00000F75:
		F_EtherCAT_VendorIDtoString := 'Gable Technologies B.V.';

	16#00000F76:
		F_EtherCAT_VendorIDtoString := 'NORCE Norwegian Research Centre AS Autonomous Systems and IoT Research Group';

	16#00000F77:
		F_EtherCAT_VendorIDtoString := 'Guangzhou Finger Technology Co.,Ltd';

	16#00000F78:
		F_EtherCAT_VendorIDtoString := 'Intercreate, Inc.';

	16#00000F79:
		F_EtherCAT_VendorIDtoString := 'Mujin, Inc.';

	16#00000F7A:
		F_EtherCAT_VendorIDtoString := 'NINGBO JANPOS TECHNOLOGY CO.,LTD';

	16#00000F7B:
		F_EtherCAT_VendorIDtoString := 'Micromega Dynamics SA';

	16#00000F7C:
		F_EtherCAT_VendorIDtoString := 'AK Optics Technology Co.,Ltd.';

	16#00000F7D:
		F_EtherCAT_VendorIDtoString := 'E3 S.r.l.';

	16#00000F7E:
		F_EtherCAT_VendorIDtoString := 'Scheidt MessTechnik';

	16#00000F80:
		F_EtherCAT_VendorIDtoString := 'Shade Technik';

	16#00000F81:
		F_EtherCAT_VendorIDtoString := 'Jeonbuk National University, College of Engineering, Department of Electronic Engineering';

	16#00000F82:
		F_EtherCAT_VendorIDtoString := 'GigaDevice Semiconductor Inc.';

	16#00000F83:
		F_EtherCAT_VendorIDtoString := 'Stellenbosch University, Faculty of Engineering, Department of Electrical and Electronic Engineering';

	16#00000F84:
		F_EtherCAT_VendorIDtoString := 'Elco Elettronica Automation s.r.l.';

	16#00000F85:
		F_EtherCAT_VendorIDtoString := 'Nanjing Rasight Intelligent Co., Ltd.';

	16#00000F86:
		F_EtherCAT_VendorIDtoString := 'KURUGANTI COMPUTERS PVT.LTD';

	16#00000F88:
		F_EtherCAT_VendorIDtoString := 'Dansk IngeniorService A/S';

	16#00000F89:
		F_EtherCAT_VendorIDtoString := 'Grapple Systems LLC';

	16#00000F8A:
		F_EtherCAT_VendorIDtoString := 'National Chung-Shan Institute of Science and Technology';

	16#00000F8B:
		F_EtherCAT_VendorIDtoString := 'FT System S.r.l. a socio unico';

	16#00000F8C:
		F_EtherCAT_VendorIDtoString := 'Stage-Kinetik Gesellschaft fur Buhnenproduktionen mbH';

	16#00000F8D:
		F_EtherCAT_VendorIDtoString := 'Shanghai Zhongchen Electronic Technology Co.,Ltd.';

	16#00000F8E:
		F_EtherCAT_VendorIDtoString := 'Eurocontrol S.p.A.';

	16#00000F8F:
		F_EtherCAT_VendorIDtoString := 'Syrma SGS Technology Ltd.';

	16#00000F90:
		F_EtherCAT_VendorIDtoString := 'Hindustan Aeronautics Limited';

	16#00000F91:
		F_EtherCAT_VendorIDtoString := 'Supercomputing Systems AG';

	16#00000F92:
		F_EtherCAT_VendorIDtoString := 'Janatics India Private Limited';

	16#00000F93:
		F_EtherCAT_VendorIDtoString := 'Carl Zeiss Spectroscopy GmbH';

	16#00000F94:
		F_EtherCAT_VendorIDtoString := 'Fullmo GmbH';

	16#00000F96:
		F_EtherCAT_VendorIDtoString := 'Shanghai Real Thread Electronic Technology Co., Ltd.';

	16#00000F97:
		F_EtherCAT_VendorIDtoString := 'Norgren Ltd';

	16#00000F98:
		F_EtherCAT_VendorIDtoString := 'Forbes Marshall Technology Pvt. Ltd.';

	16#00000F99:
		F_EtherCAT_VendorIDtoString := 'Stony Brook University, College of Engineering and Applied Sciences, Department of Electrical and Computer Engineering, Spellman High Voltage Power Electronics Lab';

	16#00000F9A:
		F_EtherCAT_VendorIDtoString := 'Guangzhou Servode Electric Co.,Ltd';

	16#00000F9B:
		F_EtherCAT_VendorIDtoString := 'Kolorrol Technologies Pvt. Ltd.';

	16#00000F9C:
		F_EtherCAT_VendorIDtoString := 'Sensirion AG';

	16#00000F9D:
		F_EtherCAT_VendorIDtoString := 'e-con Systems India Pvt Ltd';

	16#00000F9E:
		F_EtherCAT_VendorIDtoString := 'Devol Robots Sdn. Bhd.';

	16#00000F9F:
		F_EtherCAT_VendorIDtoString := 'Jiangxi Hangtong Electric Technology Co., Ltd.';

	16#00000FA0:
		F_EtherCAT_VendorIDtoString := 'KOCH Pac-Systeme GmbH';

	16#00000FA1:
		F_EtherCAT_VendorIDtoString := 'SHENZHEN OUAIDI TECHNOLOGY CO., LTD.';

	16#00000FA2:
		F_EtherCAT_VendorIDtoString := 'Ocado Innovation Limited';

	16#00000FA4:
		F_EtherCAT_VendorIDtoString := 'Agiliad Technologies Pvt Ltd';

	16#00000FA5:
		F_EtherCAT_VendorIDtoString := 'SOLO Motor Controllers S.R.L.';

	16#00000FA6:
		F_EtherCAT_VendorIDtoString := 'ZAP Surgical Systems, Inc.';

	16#00000FA7:
		F_EtherCAT_VendorIDtoString := 'SCIENTIFIC MES-TECHNIK PVT. LTD.';

	16#00000FA8:
		F_EtherCAT_VendorIDtoString := 'Briter Shenzhen Technology Co., Ltd.';

	16#00000FA9:
		F_EtherCAT_VendorIDtoString := 'US Technology International Private Limited';

	16#00000FAA:
		F_EtherCAT_VendorIDtoString := 'Human in Motion Robotics Inc.';

	16#00000FAB:
		F_EtherCAT_VendorIDtoString := 'HAGMANN TEC AG';

	16#00000FAC:
		F_EtherCAT_VendorIDtoString := 'Tortuga Agricultural Technologies, Inc dba. Tortuga AgTech';

	16#00000FAE:
		F_EtherCAT_VendorIDtoString := 'Arrow (China) Electronics Trading Co. Ltd. Shenzhen Branch';

	16#00000FAF:
		F_EtherCAT_VendorIDtoString := 'Jiangsu Hengli Hydraulic Technology Co., Ltd.';

	16#00000FB1:
		F_EtherCAT_VendorIDtoString := 'Mideker Sensor (Shanghai) Co., Ltd.';

	16#00000FB2:
		F_EtherCAT_VendorIDtoString := 'CastNX Private Limited';

	16#00000FB3:
		F_EtherCAT_VendorIDtoString := 'Herch Opto Electronic Technology Co., Ltd.';

	16#00000FB4:
		F_EtherCAT_VendorIDtoString := 'Guangdong Youbi Intelligent Equipment Technology Co., Ltd.';

	16#00000FB5:
		F_EtherCAT_VendorIDtoString := 'SAMICK PRECISION IND. CO.,LTD.';

	16#00000FB6:
		F_EtherCAT_VendorIDtoString := 'NESSAP s.r.o.';

	16#00000FB7:
		F_EtherCAT_VendorIDtoString := 'MICROPHASE s.r.l.';

	16#00000FB9:
		F_EtherCAT_VendorIDtoString := 'Efftronics System Pvt. Ltd.';

	16#00000FBA:
		F_EtherCAT_VendorIDtoString := 'Daudin Co., Ltd.';

	16#00000FBB:
		F_EtherCAT_VendorIDtoString := 'Shenzhen Faroad Intelligent Equipment Co., Ltd';

	16#00000FBC:
		F_EtherCAT_VendorIDtoString := 'YAMABISHI Corporation';

	16#00000FBD:
		F_EtherCAT_VendorIDtoString := 'Hyundai Mobis Co., Ltd.';

	16#00000FC0:
		F_EtherCAT_VendorIDtoString := 'Teckinsoft Neuronics Private Limited';

	16#00000FC1:
		F_EtherCAT_VendorIDtoString := 'IEMEIL Intelligent Technology (Zhejiang) Co., Ltd';

	16#00000FC2:
		F_EtherCAT_VendorIDtoString := 'HULL Precision Instrument Corporation';

	16#00000FC4:
		F_EtherCAT_VendorIDtoString := 'Zhejiang UTRIO Technology Co., Ltd.';

	16#00000FC6:
		F_EtherCAT_VendorIDtoString := 'Erratic di Massimo Visona';

	16#00000FC7:
		F_EtherCAT_VendorIDtoString := 'Jiangnan Yifan Motor Co., Ltd.';

	16#00000FCA:
		F_EtherCAT_VendorIDtoString := 'Flowsoft Co., Ltd.';

	16#00000FCB:
		F_EtherCAT_VendorIDtoString := 'Star Cutter Company';

	16#00000FCC:
		F_EtherCAT_VendorIDtoString := 'Celestial Oncology China Co.,LTD.';

	16#00000FCD:
		F_EtherCAT_VendorIDtoString := 'Dotwil RF (Anhui) Technology Co., Ltd.';

	16#00000FCE:
		F_EtherCAT_VendorIDtoString := 'KIKUSUI ELECTRONICS CORP.';

	16#00000FCF:
		F_EtherCAT_VendorIDtoString := 'Cognitive Photonics (Beijing) Laser Technology Co., Ltd.';

	16#00000FD1:
		F_EtherCAT_VendorIDtoString := 'Mo Chi Industrial Co., LTD.';

	16#00000FD2:
		F_EtherCAT_VendorIDtoString := 'Shanghai Insky Intelligent Technology Co., Ltd.';

	16#00000FD3:
		F_EtherCAT_VendorIDtoString := 'ELDAPS Technology Solutions Private Limited';

	16#00000FD4:
		F_EtherCAT_VendorIDtoString := 'HL Mando Corp.';

	16#00000FD5:
		F_EtherCAT_VendorIDtoString := 'Adeeb Robotics LLC';

	16#00000FD6:
		F_EtherCAT_VendorIDtoString := 'Xian Actionpower Electric Co., Ltd.';

	16#00000FD7:
		F_EtherCAT_VendorIDtoString := 'YanCi Machinery Technology Research (Dalian) Co., Ltd.';

	16#00000FD8:
		F_EtherCAT_VendorIDtoString := 'Xiaomi EV Technology Co., Ltd.';

	16#00000FD9:
		F_EtherCAT_VendorIDtoString := 'Carl Zeiss Meditec AG';

	16#00000FDA:
		F_EtherCAT_VendorIDtoString := 'ITronic Meres- es Automatizalas Technikai Kft.';

	16#00000FDB:
		F_EtherCAT_VendorIDtoString := 'Cincinnati Incorporated';

	16#00000FDC:
		F_EtherCAT_VendorIDtoString := 'Shanghai Erchuan CNC Technology (Group) Co., Ltd.';

	16#00000FDD:
		F_EtherCAT_VendorIDtoString := 'Center for Astrophysics | Harvard & Smithsonian, Smithsonian Astrophysical Observatory';

	16#00000FDE:
		F_EtherCAT_VendorIDtoString := 'AnTronix GmbH';

	16#00000FDF:
		F_EtherCAT_VendorIDtoString := 'SuninCNS, Inc.';

	16#00000FE0:
		F_EtherCAT_VendorIDtoString := 'Leroy Automation';

	16#00000FE1:
		F_EtherCAT_VendorIDtoString := 'Zap Energy Inc.';

	16#00000FE3:
		F_EtherCAT_VendorIDtoString := 'A&DS Co., Ltd.';

	16#00000FE4:
		F_EtherCAT_VendorIDtoString := 'Simple Intelligence Technology (Shanghai) Co., Ltd.';

	16#00000FE5:
		F_EtherCAT_VendorIDtoString := 'Shenzhen Huihe Technology Co.LTD';

